ABB RobotStudio station: Laboratorio 1 RS.rspag

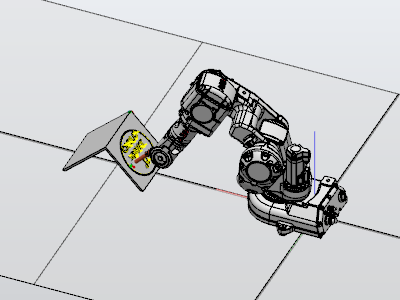
--- station ---
Station Laboratorio 1 RS (saved by RobotStudio 23.2.10395.0)
Controller IRB140_6_81, task T_ROB1: task frame (RAPID world) sits at (164.79, 0, 0) mm in the station
Controller IRB140_6_81
  mechanical unit ROB_1: IRB140_6_81_C_03, 6 joints, base frame (0, 0, 0) mm
Layout (positions relative to the parent item):
  - IRB140_6_81_C_03 [mechanism, from %ABB.RobotStudio.Models.IRB140%\IRB140_6_81_C_G_03.rslib] at (164.79, 0, 0) mm; joint values [0.1988, 0.9588, 0.0809, 3.4211, 0.7525, 2.9948] (rad or m)
  - Tableros [part] at (1000, 0, 0) mm, rotated rx 90 ry 0 rz 180 deg, size 410.4 x 204.7 x 300 mm
  - Marcador [mechanism] at (773, 110, 211.85) mm, rotated rx -180 ry 72.73 rz -180 deg
      TCP MarcadorTCP at (65.54, 0, 135.85) mm, rotated rx 0 ry 25.76 rz 0 deg
      links: EnsambleToolMarcador_3
Attachment: Marcador is attached to IRB140_6_81_C_03 / Link6
Targets, tools, work objects and paths stored in the station and not in the controller backup, written as RAPID:
! task T_ROB1
MODULE Module1
  CONST robtarget Target_350:=[[69.849,197.313,-20],[1,0,0,0],[0,0,0,0],[9E+09,9E+09,9E+09,9E+09,9E+09,9E+09]];
  CONST robtarget Target_360:=[[69.849,197.313,0],[1,0,0,0],[0,0,0,0],[9E+09,9E+09,9E+09,9E+09,9E+09,9E+09]];
  CONST robtarget Target_370:=[[68.877,199.4,0],[1,0,0,0],[0,0,0,0],[9E+09,9E+09,9E+09,9E+09,9E+09,9E+09]];
  CONST robtarget Target_380:=[[67.982,201.773,0],[1,0,0,0],[0,0,0,0],[9E+09,9E+09,9E+09,9E+09,9E+09,9E+09]];
  CONST robtarget Target_390:=[[67.399,204.703,0],[1,0,0,0],[0,0,0,0],[9E+09,9E+09,9E+09,9E+09,9E+09,9E+09]];
  CONST robtarget Target_400:=[[67.178,208.126,0],[1,0,0,0],[0,0,0,0],[9E+09,9E+09,9E+09,9E+09,9E+09,9E+09]];
  CONST robtarget Target_410:=[[71.703,219.575,0],[1,0,0,0],[0,0,0,0],[9E+09,9E+09,9E+09,9E+09,9E+09,9E+09]];
  CONST robtarget Target_420:=[[83.827,223.815,0],[1,0,0,0],[0,0,0,0],[9E+09,9E+09,9E+09,9E+09,9E+09,9E+09]];
  CONST robtarget Target_430:=[[96.066,219.588,0],[1,0,0,0],[0,0,0,0],[9E+09,9E+09,9E+09,9E+09,9E+09,9E+09]];
  CONST robtarget Target_440:=[[100.423,208.152,0],[1,0,0,0],[0,0,0,0],[9E+09,9E+09,9E+09,9E+09,9E+09,9E+09]];
  CONST robtarget Target_450:=[[100.19,204.561,0],[1,0,0,0],[0,0,0,0],[9E+09,9E+09,9E+09,9E+09,9E+09,9E+09]];
  CONST robtarget Target_460:=[[99.489,201.747,0],[1,0,0,0],[0,0,0,0],[9E+09,9E+09,9E+09,9E+09,9E+09,9E+09]];
  CONST robtarget Target_470:=[[98.608,199.348,0],[1,0,0,0],[0,0,0,0],[9E+09,9E+09,9E+09,9E+09,9E+09,9E+09]];
  CONST robtarget Target_480:=[[97.674,197.313,0],[1,0,0,0],[0,0,0,0],[9E+09,9E+09,9E+09,9E+09,9E+09,9E+09]];
  CONST robtarget Target_490:=[[90.154,197.313,0],[1,0,0,0],[0,0,0,0],[9E+09,9E+09,9E+09,9E+09,9E+09,9E+09]];
  CONST robtarget Target_500:=[[90.154,198.039,0],[1,0,0,0],[0,0,0,0],[9E+09,9E+09,9E+09,9E+09,9E+09,9E+09]];
  CONST robtarget Target_510:=[[91.386,199.452,0],[1,0,0,0],[0,0,0,0],[9E+09,9E+09,9E+09,9E+09,9E+09,9E+09]];
  CONST robtarget Target_520:=[[92.721,201.358,0],[1,0,0,0],[0,0,0,0],[9E+09,9E+09,9E+09,9E+09,9E+09,9E+09]];
  CONST robtarget Target_530:=[[93.901,203.783,0],[1,0,0,0],[0,0,0,0],[9E+09,9E+09,9E+09,9E+09,9E+09,9E+09]];
  CONST robtarget Target_540:=[[94.433,206.804,0],[1,0,0,0],[0,0,0,0],[9E+09,9E+09,9E+09,9E+09,9E+09,9E+09]];
  CONST robtarget Target_550:=[[93.901,209.864,0],[1,0,0,0],[0,0,0,0],[9E+09,9E+09,9E+09,9E+09,9E+09,9E+09]];
  CONST robtarget Target_560:=[[92.151,212.639,0],[1,0,0,0],[0,0,0,0],[9E+09,9E+09,9E+09,9E+09,9E+09,9E+09]];
  CONST robtarget Target_570:=[[88.87,214.726,0],[1,0,0,0],[0,0,0,0],[9E+09,9E+09,9E+09,9E+09,9E+09,9E+09]];
  CONST robtarget Target_580:=[[83.852,215.517,0],[1,0,0,0],[0,0,0,0],[9E+09,9E+09,9E+09,9E+09,9E+09,9E+09]];
  CONST robtarget Target_590:=[[78.938,214.752,0],[1,0,0,0],[0,0,0,0],[9E+09,9E+09,9E+09,9E+09,9E+09,9E+09]];
  CONST robtarget Target_600:=[[75.632,212.794,0],[1,0,0,0],[0,0,0,0],[9E+09,9E+09,9E+09,9E+09,9E+09,9E+09]];
  CONST robtarget Target_610:=[[73.713,210.032,0],[1,0,0,0],[0,0,0,0],[9E+09,9E+09,9E+09,9E+09,9E+09,9E+09]];
  CONST robtarget Target_620:=[[73.169,206.856,0],[1,0,0,0],[0,0,0,0],[9E+09,9E+09,9E+09,9E+09,9E+09,9E+09]];
  CONST robtarget Target_630:=[[73.648,204.042,0],[1,0,0,0],[0,0,0,0],[9E+09,9E+09,9E+09,9E+09,9E+09,9E+09]];
  CONST robtarget Target_640:=[[74.828,201.592,0],[1,0,0,0],[0,0,0,0],[9E+09,9E+09,9E+09,9E+09,9E+09,9E+09]];
  CONST robtarget Target_650:=[[76.228,199.595,0],[1,0,0,0],[0,0,0,0],[9E+09,9E+09,9E+09,9E+09,9E+09,9E+09]];
  CONST robtarget Target_660:=[[77.473,198.117,0],[1,0,0,0],[0,0,0,0],[9E+09,9E+09,9E+09,9E+09,9E+09,9E+09]];
  CONST robtarget Target_670:=[[77.473,197.313,0],[1,0,0,0],[0,0,0,0],[9E+09,9E+09,9E+09,9E+09,9E+09,9E+09]];
  CONST robtarget Target_680:=[[69.849,197.313,0],[1,0,0,0],[0,0,0,0],[9E+09,9E+09,9E+09,9E+09,9E+09,9E+09]];
  CONST robtarget Target_690:=[[69.849,197.313,-40],[1,0,0,0],[0,0,0,0],[9E+09,9E+09,9E+09,9E+09,9E+09,9E+09]];
  CONST robtarget Target_850:=[[99.801,165.624,-20],[1,0,0,0],[0,0,0,0],[9E+09,9E+09,9E+09,9E+09,9E+09,9E+09]];
  CONST robtarget Target_860:=[[99.801,165.624,0],[1,0,0,0],[0,0,0,0],[9E+09,9E+09,9E+09,9E+09,9E+09,9E+09]];
  CONST robtarget Target_870:=[[67.801,176.438,0],[1,0,0,0],[0,0,0,0],[9E+09,9E+09,9E+09,9E+09,9E+09,9E+09]];
  CONST robtarget Target_880:=[[67.801,185.203,0],[1,0,0,0],[0,0,0,0],[9E+09,9E+09,9E+09,9E+09,9E+09,9E+09]];
  CONST robtarget Target_890:=[[99.801,196.016,0],[1,0,0,0],[0,0,0,0],[9E+09,9E+09,9E+09,9E+09,9E+09,9E+09]];
  CONST robtarget Target_900:=[[99.801,187.977,0],[1,0,0,0],[0,0,0,0],[9E+09,9E+09,9E+09,9E+09,9E+09,9E+09]];
  CONST robtarget Target_910:=[[93.266,185.955,0],[1,0,0,0],[0,0,0,0],[9E+09,9E+09,9E+09,9E+09,9E+09,9E+09]];
  CONST robtarget Target_920:=[[93.266,175.893,0],[1,0,0,0],[0,0,0,0],[9E+09,9E+09,9E+09,9E+09,9E+09,9E+09]];
  CONST robtarget Target_930:=[[99.801,173.896,0],[1,0,0,0],[0,0,0,0],[9E+09,9E+09,9E+09,9E+09,9E+09,9E+09]];
  CONST robtarget Target_940:=[[99.801,165.624,0],[1,0,0,0],[0,0,0,0],[9E+09,9E+09,9E+09,9E+09,9E+09,9E+09]];
  CONST robtarget Target_950:=[[87.457,177.656,-20],[1,0,0,0],[0,0,0,0],[9E+09,9E+09,9E+09,9E+09,9E+09,9E+09]];
  CONST robtarget Target_960:=[[87.457,177.656,0],[1,0,0,0],[0,0,0,0],[9E+09,9E+09,9E+09,9E+09,9E+09,9E+09]];
  CONST robtarget Target_970:=[[76.877,180.924,0],[1,0,0,0],[0,0,0,0],[9E+09,9E+09,9E+09,9E+09,9E+09,9E+09]];
  CONST robtarget Target_980:=[[87.457,184.217,0],[1,0,0,0],[0,0,0,0],[9E+09,9E+09,9E+09,9E+09,9E+09,9E+09]];
  CONST robtarget Target_990:=[[87.457,177.656,0],[1,0,0,0],[0,0,0,0],[9E+09,9E+09,9E+09,9E+09,9E+09,9E+09]];
  CONST robtarget Target_1000:=[[87.457,177.656,-20],[1,0,0,0],[0,0,0,0],[9E+09,9E+09,9E+09,9E+09,9E+09,9E+09]];
  CONST robtarget Target_1010:=[[99.801,132.872,-20],[1,0,0,0],[0,0,0,0],[9E+09,9E+09,9E+09,9E+09,9E+09,9E+09]];
  CONST robtarget Target_1020:=[[99.801,132.872,0],[1,0,0,0],[0,0,0,0],[9E+09,9E+09,9E+09,9E+09,9E+09,9E+09]];
  CONST robtarget Target_1030:=[[86.186,143.634,0],[1,0,0,0],[0,0,0,0],[9E+09,9E+09,9E+09,9E+09,9E+09,9E+09]];
  CONST robtarget Target_1040:=[[82.543,139.199,0],[1,0,0,0],[0,0,0,0],[9E+09,9E+09,9E+09,9E+09,9E+09,9E+09]];
  CONST robtarget Target_1050:=[[76.592,137.54,0],[1,0,0,0],[0,0,0,0],[9E+09,9E+09,9E+09,9E+09,9E+09,9E+09]];
  CONST robtarget Target_1060:=[[72.3,138.551,0],[1,0,0,0],[0,0,0,0],[9E+09,9E+09,9E+09,9E+09,9E+09,9E+09]];
  CONST robtarget Target_1070:=[[69.512,141.274,0],[1,0,0,0],[0,0,0,0],[9E+09,9E+09,9E+09,9E+09,9E+09,9E+09]];
  CONST robtarget Target_1080:=[[68.138,144.93,0],[1,0,0,0],[0,0,0,0],[9E+09,9E+09,9E+09,9E+09,9E+09,9E+09]];
  CONST robtarget Target_1090:=[[67.801,149.572,0],[1,0,0,0],[0,0,0,0],[9E+09,9E+09,9E+09,9E+09,9E+09,9E+09]];
  CONST robtarget Target_1100:=[[67.801,162.434,0],[1,0,0,0],[0,0,0,0],[9E+09,9E+09,9E+09,9E+09,9E+09,9E+09]];
  CONST robtarget Target_1110:=[[99.801,162.434,0],[1,0,0,0],[0,0,0,0],[9E+09,9E+09,9E+09,9E+09,9E+09,9E+09]];
  CONST robtarget Target_1120:=[[99.801,154.447,0],[1,0,0,0],[0,0,0,0],[9E+09,9E+09,9E+09,9E+09,9E+09,9E+09]];
  CONST robtarget Target_1130:=[[88.053,154.447,0],[1,0,0,0],[0,0,0,0],[9E+09,9E+09,9E+09,9E+09,9E+09,9E+09]];
  CONST robtarget Target_1140:=[[88.053,151.543,0],[1,0,0,0],[0,0,0,0],[9E+09,9E+09,9E+09,9E+09,9E+09,9E+09]];
  CONST robtarget Target_1150:=[[99.801,142.648,0],[1,0,0,0],[0,0,0,0],[9E+09,9E+09,9E+09,9E+09,9E+09,9E+09]];
  CONST robtarget Target_1160:=[[99.801,132.872,0],[1,0,0,0],[0,0,0,0],[9E+09,9E+09,9E+09,9E+09,9E+09,9E+09]];
  CONST robtarget Target_1170:=[[82.297,154.447,-20],[1,0,0,0],[0,0,0,0],[9E+09,9E+09,9E+09,9E+09,9E+09,9E+09]];
  CONST robtarget Target_1180:=[[82.297,154.447,0],[1,0,0,0],[0,0,0,0],[9E+09,9E+09,9E+09,9E+09,9E+09,9E+09]];
  CONST robtarget Target_1190:=[[82.297,152.139,0],[1,0,0,0],[0,0,0,0],[9E+09,9E+09,9E+09,9E+09,9E+09,9E+09]];
  CONST robtarget Target_1200:=[[82.089,149.3,0],[1,0,0,0],[0,0,0,0],[9E+09,9E+09,9E+09,9E+09,9E+09,9E+09]];
  CONST robtarget Target_1210:=[[81.233,147.316,0],[1,0,0,0],[0,0,0,0],[9E+09,9E+09,9E+09,9E+09,9E+09,9E+09]];
  CONST robtarget Target_1220:=[[79.781,146.162,0],[1,0,0,0],[0,0,0,0],[9E+09,9E+09,9E+09,9E+09,9E+09,9E+09]];
  CONST robtarget Target_1230:=[[77.603,145.786,0],[1,0,0,0],[0,0,0,0],[9E+09,9E+09,9E+09,9E+09,9E+09,9E+09]];
  CONST robtarget Target_1240:=[[75.515,146.253,0],[1,0,0,0],[0,0,0,0],[9E+09,9E+09,9E+09,9E+09,9E+09,9E+09]];
  CONST robtarget Target_1250:=[[74.18,147.783,0],[1,0,0,0],[0,0,0,0],[9E+09,9E+09,9E+09,9E+09,9E+09,9E+09]];
  CONST robtarget Target_1260:=[[73.778,149.455,0],[1,0,0,0],[0,0,0,0],[9E+09,9E+09,9E+09,9E+09,9E+09,9E+09]];
  CONST robtarget Target_1270:=[[73.687,151.75,0],[1,0,0,0],[0,0,0,0],[9E+09,9E+09,9E+09,9E+09,9E+09,9E+09]];
  CONST robtarget Target_1280:=[[73.687,154.447,0],[1,0,0,0],[0,0,0,0],[9E+09,9E+09,9E+09,9E+09,9E+09,9E+09]];
  CONST robtarget Target_1290:=[[82.297,154.447,0],[1,0,0,0],[0,0,0,0],[9E+09,9E+09,9E+09,9E+09,9E+09,9E+09]];
  CONST robtarget Target_1300:=[[82.297,154.447,-20],[1,0,0,0],[0,0,0,0],[9E+09,9E+09,9E+09,9E+09,9E+09,9E+09]];
  CONST robtarget Target_1310:=[[99.801,109.144,-20],[1,0,0,0],[0,0,0,0],[9E+09,9E+09,9E+09,9E+09,9E+09,9E+09]];
  CONST robtarget Target_1320:=[[99.801,109.144,0],[1,0,0,0],[0,0,0,0],[9E+09,9E+09,9E+09,9E+09,9E+09,9E+09]];
  CONST robtarget Target_1330:=[[93.707,109.144,0],[1,0,0,0],[0,0,0,0],[9E+09,9E+09,9E+09,9E+09,9E+09,9E+09]];
  CONST robtarget Target_1340:=[[93.707,122.447,0],[1,0,0,0],[0,0,0,0],[9E+09,9E+09,9E+09,9E+09,9E+09,9E+09]];
  CONST robtarget Target_1350:=[[67.801,122.447,0],[1,0,0,0],[0,0,0,0],[9E+09,9E+09,9E+09,9E+09,9E+09,9E+09]];
  CONST robtarget Target_1360:=[[67.801,130.486,0],[1,0,0,0],[0,0,0,0],[9E+09,9E+09,9E+09,9E+09,9E+09,9E+09]];
  CONST robtarget Target_1370:=[[99.801,130.486,0],[1,0,0,0],[0,0,0,0],[9E+09,9E+09,9E+09,9E+09,9E+09,9E+09]];
  CONST robtarget Target_1380:=[[99.801,109.144,0],[1,0,0,0],[0,0,0,0],[9E+09,9E+09,9E+09,9E+09,9E+09,9E+09]];
  CONST robtarget Target_1390:=[[99.801,109.144,-20],[1,0,0,0],[0,0,0,0],[9E+09,9E+09,9E+09,9E+09,9E+09,9E+09]];
  CONST robtarget Target_1400:=[[83.801,76.185,-20],[1,0,0,0],[0,0,0,0],[9E+09,9E+09,9E+09,9E+09,9E+09,9E+09]];
  CONST robtarget Target_1410:=[[83.801,76.185,0],[1,0,0,0],[0,0,0,0],[9E+09,9E+09,9E+09,9E+09,9E+09,9E+09]];
  CONST robtarget Target_1420:=[[96.028,80.334,0],[1,0,0,0],[0,0,0,0],[9E+09,9E+09,9E+09,9E+09,9E+09,9E+09]];
  CONST robtarget Target_1430:=[[100.475,91.692,0],[1,0,0,0],[0,0,0,0],[9E+09,9E+09,9E+09,9E+09,9E+09,9E+09]];
  CONST robtarget Target_1440:=[[95.976,103.05,0],[1,0,0,0],[0,0,0,0],[9E+09,9E+09,9E+09,9E+09,9E+09,9E+09]];
  CONST robtarget Target_1450:=[[83.801,107.173,0],[1,0,0,0],[0,0,0,0],[9E+09,9E+09,9E+09,9E+09,9E+09,9E+09]];
  CONST robtarget Target_1460:=[[71.613,103.05,0],[1,0,0,0],[0,0,0,0],[9E+09,9E+09,9E+09,9E+09,9E+09,9E+09]];
  CONST robtarget Target_1470:=[[67.126,91.692,0],[1,0,0,0],[0,0,0,0],[9E+09,9E+09,9E+09,9E+09,9E+09,9E+09]];
  CONST robtarget Target_1480:=[[71.587,80.334,0],[1,0,0,0],[0,0,0,0],[9E+09,9E+09,9E+09,9E+09,9E+09,9E+09]];
  CONST robtarget Target_1490:=[[83.801,76.185,0],[1,0,0,0],[0,0,0,0],[9E+09,9E+09,9E+09,9E+09,9E+09,9E+09]];
  CONST robtarget Target_1500:=[[75.58,96.671,-20],[1,0,0,0],[0,0,0,0],[9E+09,9E+09,9E+09,9E+09,9E+09,9E+09]];
  CONST robtarget Target_1510:=[[75.58,96.671,0],[1,0,0,0],[0,0,0,0],[9E+09,9E+09,9E+09,9E+09,9E+09,9E+09]];
  CONST robtarget Target_1520:=[[78.887,98.266,0],[1,0,0,0],[0,0,0,0],[9E+09,9E+09,9E+09,9E+09,9E+09,9E+09]];
  CONST robtarget Target_1530:=[[83.801,98.875,0],[1,0,0,0],[0,0,0,0],[9E+09,9E+09,9E+09,9E+09,9E+09,9E+09]];
  CONST robtarget Target_1540:=[[88.702,98.292,0],[1,0,0,0],[0,0,0,0],[9E+09,9E+09,9E+09,9E+09,9E+09,9E+09]];
  CONST robtarget Target_1550:=[[91.969,96.697,0],[1,0,0,0],[0,0,0,0],[9E+09,9E+09,9E+09,9E+09,9E+09,9E+09]];
  CONST robtarget Target_1560:=[[93.862,94.376,0],[1,0,0,0],[0,0,0,0],[9E+09,9E+09,9E+09,9E+09,9E+09,9E+09]];
  CONST robtarget Target_1570:=[[94.433,91.666,0],[1,0,0,0],[0,0,0,0],[9E+09,9E+09,9E+09,9E+09,9E+09,9E+09]];
  CONST robtarget Target_1580:=[[93.823,88.917,0],[1,0,0,0],[0,0,0,0],[9E+09,9E+09,9E+09,9E+09,9E+09,9E+09]];
  CONST robtarget Target_1590:=[[91.917,86.635,5],[1,0,0,0],[0,0,0,0],[9E+09,9E+09,9E+09,9E+09,9E+09,9E+09]];
  CONST robtarget Target_1600:=[[88.663,85.041,0],[1,0,0,0],[0,0,0,0],[9E+09,9E+09,9E+09,9E+09,9E+09,9E+09]];
  CONST robtarget Target_1610:=[[83.801,84.483,0],[1,0,0,0],[0,0,0,0],[9E+09,9E+09,9E+09,9E+09,9E+09,9E+09]];
  CONST robtarget Target_1620:=[[78.912,85.066,0],[1,0,0,0],[0,0,0,0],[9E+09,9E+09,9E+09,9E+09,9E+09,9E+09]];
  CONST robtarget Target_1630:=[[75.632,86.661,0],[1,0,0,0],[0,0,0,0],[9E+09,9E+09,9E+09,9E+09,9E+09,9E+09]];
  CONST robtarget Target_1640:=[[73.739,88.969,0],[1,0,0,0],[0,0,0,0],[9E+09,9E+09,9E+09,9E+09,9E+09,9E+09]];
  CONST robtarget Target_1650:=[[73.169,91.666,0],[1,0,0,0],[0,0,0,0],[9E+09,9E+09,9E+09,9E+09,9E+09,9E+09]];
  CONST robtarget Target_1660:=[[73.7,94.35,0],[1,0,0,0],[0,0,0,0],[9E+09,9E+09,9E+09,9E+09,9E+09,9E+09]];
  CONST robtarget Target_1670:=[[75.58,96.671,0],[1,0,0,0],[0,0,0,0],[9E+09,9E+09,9E+09,9E+09,9E+09,9E+09]];
  CONST robtarget Target_1680:=[[75.58,96.671,-20],[1,0,0,0],[0,0,0,0],[9E+09,9E+09,9E+09,9E+09,9E+09,9E+09]];
  CONST robtarget Target_1690:=[[120.488,219.705,-20],[1,0,0,0],[0,0,0,0],[9E+09,9E+09,9E+09,9E+09,9E+09,9E+09]];
  CONST robtarget Target_1700:=[[120.488,219.705,0],[1,0,0,0],[0,0,0,0],[9E+09,9E+09,9E+09,9E+09,9E+09,9E+09]];
  CONST robtarget Target_1710:=[[120.488,204.353,0],[1,0,0,0],[0,0,0,0],[9E+09,9E+09,9E+09,9E+09,9E+09,9E+09]];
  CONST robtarget Target_1720:=[[143.1,204.353,0.001],[1,0,0,0],[0,0,0,0],[9E+09,9E+09,9E+09,9E+09,9E+09,9E+09]];
  CONST robtarget Target_1730:=[[147.016,205.066,0.001],[1,0,0,0],[0,0,0,0],[9E+09,9E+09,9E+09,9E+09,9E+09,9E+09]];
  CONST robtarget Target_1740:=[[150.154,207.206,0.001],[1,0,0,0],[0,0,0,0],[9E+09,9E+09,9E+09,9E+09,9E+09,9E+09]];
  CONST robtarget Target_1750:=[[152.293,211.005,0.001],[1,0,0,0],[0,0,0,0],[9E+09,9E+09,9E+09,9E+09,9E+09,9E+09]];
  CONST robtarget Target_1760:=[[152.98,216.049,0.001],[1,0,0,0],[0,0,0,0],[9E+09,9E+09,9E+09,9E+09,9E+09,9E+09]];
  CONST robtarget Target_1770:=[[152.825,220.042,0.001],[1,0,0,0],[0,0,0,0],[9E+09,9E+09,9E+09,9E+09,9E+09,9E+09]];
  CONST robtarget Target_1780:=[[152.358,223.335,0.001],[1,0,0,0],[0,0,0,0],[9E+09,9E+09,9E+09,9E+09,9E+09,9E+09]];
  CONST robtarget Target_1790:=[[145.875,223.335,0.001],[1,0,0,0],[0,0,0,0],[9E+09,9E+09,9E+09,9E+09,9E+09,9E+09]];
  CONST robtarget Target_1800:=[[146.601,220.6,0.001],[1,0,0,0],[0,0,0,0],[9E+09,9E+09,9E+09,9E+09,9E+09,9E+09]];
  CONST robtarget Target_1810:=[[146.938,217.89,0.001],[1,0,0,0],[0,0,0,0],[9E+09,9E+09,9E+09,9E+09,9E+09,9E+09]];
  CONST robtarget Target_1820:=[[146.342,214.609,0.001],[1,0,0,0],[0,0,0,0],[9E+09,9E+09,9E+09,9E+09,9E+09,9E+09]];
  CONST robtarget Target_1830:=[[144.656,212.989,0.001],[1,0,0,0],[0,0,0,0],[9E+09,9E+09,9E+09,9E+09,9E+09,9E+09]];
  CONST robtarget Target_1840:=[[142.219,212.444,0.001],[1,0,0,0],[0,0,0,0],[9E+09,9E+09,9E+09,9E+09,9E+09,9E+09]];
  CONST robtarget Target_1850:=[[139.133,212.392,0],[1,0,0,0],[0,0,0,0],[9E+09,9E+09,9E+09,9E+09,9E+09,9E+09]];
  CONST robtarget Target_1860:=[[126.297,212.392,0],[1,0,0,0],[0,0,0,0],[9E+09,9E+09,9E+09,9E+09,9E+09,9E+09]];
  CONST robtarget Target_1870:=[[126.297,219.705,0],[1,0,0,0],[0,0,0,0],[9E+09,9E+09,9E+09,9E+09,9E+09,9E+09]];
  CONST robtarget Target_1880:=[[120.488,219.705,0],[1,0,0,0],[0,0,0,0],[9E+09,9E+09,9E+09,9E+09,9E+09,9E+09]];
  CONST robtarget Target_1890:=[[120.488,219.705,-20],[1,0,0,0],[0,0,0,0],[9E+09,9E+09,9E+09,9E+09,9E+09,9E+09]];
  CONST robtarget Target_1900:=[[153.162,184.515,-20],[1,0,0,0],[0,0,0,0],[9E+09,9E+09,9E+09,9E+09,9E+09,9E+09]];
  CONST robtarget Target_1910:=[[153.162,184.515,0],[1,0,0,0],[0,0,0,0],[9E+09,9E+09,9E+09,9E+09,9E+09,9E+09]];
  CONST robtarget Target_1920:=[[148.715,173.157,0.001],[1,0,0,0],[0,0,0,0],[9E+09,9E+09,9E+09,9E+09,9E+09,9E+09]];
  CONST robtarget Target_1930:=[[136.488,169.008,0],[1,0,0,0],[0,0,0,0],[9E+09,9E+09,9E+09,9E+09,9E+09,9E+09]];
  CONST robtarget Target_1940:=[[124.274,173.157,0],[1,0,0,0],[0,0,0,0],[9E+09,9E+09,9E+09,9E+09,9E+09,9E+09]];
  CONST robtarget Target_1950:=[[119.814,184.515,0],[1,0,0,0],[0,0,0,0],[9E+09,9E+09,9E+09,9E+09,9E+09,9E+09]];
  CONST robtarget Target_1960:=[[124.3,195.874,0],[1,0,0,0],[0,0,0,0],[9E+09,9E+09,9E+09,9E+09,9E+09,9E+09]];
  CONST robtarget Target_1970:=[[136.488,199.997,0],[1,0,0,0],[0,0,0,0],[9E+09,9E+09,9E+09,9E+09,9E+09,9E+09]];
  CONST robtarget Target_1980:=[[148.663,195.874,0.001],[1,0,0,0],[0,0,0,0],[9E+09,9E+09,9E+09,9E+09,9E+09,9E+09]];
  CONST robtarget Target_1990:=[[153.162,184.515,0.001],[1,0,0,0],[0,0,0,0],[9E+09,9E+09,9E+09,9E+09,9E+09,9E+09]];
  CONST robtarget Target_2000:=[[144.604,179.459,-20],[1,0,0,0],[0,0,0,0],[9E+09,9E+09,9E+09,9E+09,9E+09,9E+09]];
  CONST robtarget Target_2010:=[[144.604,179.459,0.001],[1,0,0,0],[0,0,0,0],[9E+09,9E+09,9E+09,9E+09,9E+09,9E+09]];
  CONST robtarget Target_2020:=[[141.35,177.864,0.001],[1,0,0,0],[0,0,0,0],[9E+09,9E+09,9E+09,9E+09,9E+09,9E+09]];
  CONST robtarget Target_2030:=[[136.488,177.306,0],[1,0,0,0],[0,0,0,0],[9E+09,9E+09,9E+09,9E+09,9E+09,9E+09]];
  CONST robtarget Target_2040:=[[131.6,177.89,0],[1,0,0,0],[0,0,0,0],[9E+09,9E+09,9E+09,9E+09,9E+09,9E+09]];
  CONST robtarget Target_2050:=[[128.319,179.485,0],[1,0,0,0],[0,0,0,0],[9E+09,9E+09,9E+09,9E+09,9E+09,9E+09]];
  CONST robtarget Target_2060:=[[126.426,181.793,0],[1,0,0,0],[0,0,0,0],[9E+09,9E+09,9E+09,9E+09,9E+09,9E+09]];
  CONST robtarget Target_2070:=[[125.856,184.489,0],[1,0,0,0],[0,0,0,0],[9E+09,9E+09,9E+09,9E+09,9E+09,9E+09]];
  CONST robtarget Target_2080:=[[126.387,187.173,0],[1,0,0,0],[0,0,0,0],[9E+09,9E+09,9E+09,9E+09,9E+09,9E+09]];
  CONST robtarget Target_2090:=[[128.267,189.494,0],[1,0,0,0],[0,0,0,0],[9E+09,9E+09,9E+09,9E+09,9E+09,9E+09]];
  CONST robtarget Target_2100:=[[131.574,191.089,0],[1,0,0,0],[0,0,0,0],[9E+09,9E+09,9E+09,9E+09,9E+09,9E+09]];
  CONST robtarget Target_2110:=[[136.488,191.699,0],[1,0,0,0],[0,0,0,0],[9E+09,9E+09,9E+09,9E+09,9E+09,9E+09]];
  CONST robtarget Target_2120:=[[141.389,191.115,0.001],[1,0,0,0],[0,0,0,0],[9E+09,9E+09,9E+09,9E+09,9E+09,9E+09]];
  CONST robtarget Target_2130:=[[144.656,189.52,0.001],[1,0,0,0],[0,0,0,0],[9E+09,9E+09,9E+09,9E+09,9E+09,9E+09]];
  CONST robtarget Target_2140:=[[146.549,187.199,0.001],[1,0,0,0],[0,0,0,0],[9E+09,9E+09,9E+09,9E+09,9E+09,9E+09]];
  CONST robtarget Target_2150:=[[147.12,184.489,0.001],[1,0,0,0],[0,0,0,0],[9E+09,9E+09,9E+09,9E+09,9E+09,9E+09]];
  CONST robtarget Target_2160:=[[146.51,181.741,0.001],[1,0,0,0],[0,0,0,0],[9E+09,9E+09,9E+09,9E+09,9E+09,9E+09]];
  CONST robtarget Target_2170:=[[144.604,179.459,0.001],[1,0,0,0],[0,0,0,0],[9E+09,9E+09,9E+09,9E+09,9E+09,9E+09]];
  CONST robtarget Target_2180:=[[144.604,179.459,-20],[1,0,0,0],[0,0,0,0],[9E+09,9E+09,9E+09,9E+09,9E+09,9E+09]];
  CONST robtarget Target_2190:=[[152.488,136.827,-20],[1,0,0,0],[0,0,0,0],[9E+09,9E+09,9E+09,9E+09,9E+09,9E+09]];
  CONST robtarget Target_2200:=[[152.488,136.827,0.001],[1,0,0,0],[0,0,0,0],[9E+09,9E+09,9E+09,9E+09,9E+09,9E+09]];
  CONST robtarget Target_2210:=[[120.488,136.827,0],[1,0,0,0],[0,0,0,0],[9E+09,9E+09,9E+09,9E+09,9E+09,9E+09]];
  CONST robtarget Target_2220:=[[120.488,144.165,0],[1,0,0,0],[0,0,0,0],[9E+09,9E+09,9E+09,9E+09,9E+09,9E+09]];
  CONST robtarget Target_2230:=[[138.822,144.165,0],[1,0,0,0],[0,0,0,0],[9E+09,9E+09,9E+09,9E+09,9E+09,9E+09]];
  CONST robtarget Target_2240:=[[120.488,154.382,0],[1,0,0,0],[0,0,0,0],[9E+09,9E+09,9E+09,9E+09,9E+09,9E+09]];
  CONST robtarget Target_2250:=[[120.488,164.237,0],[1,0,0,0],[0,0,0,0],[9E+09,9E+09,9E+09,9E+09,9E+09,9E+09]];
  CONST robtarget Target_2260:=[[152.488,164.237,0.001],[1,0,0,0],[0,0,0,0],[9E+09,9E+09,9E+09,9E+09,9E+09,9E+09]];
  CONST robtarget Target_2270:=[[152.488,156.898,0.001],[1,0,0,0],[0,0,0,0],[9E+09,9E+09,9E+09,9E+09,9E+09,9E+09]];
  CONST robtarget Target_2280:=[[130.186,156.898,0],[1,0,0,0],[0,0,0,0],[9E+09,9E+09,9E+09,9E+09,9E+09,9E+09]];
  CONST robtarget Target_2290:=[[152.488,144.554,0.001],[1,0,0,0],[0,0,0,0],[9E+09,9E+09,9E+09,9E+09,9E+09,9E+09]];
  CONST robtarget Target_2300:=[[152.488,136.827,0.001],[1,0,0,0],[0,0,0,0],[9E+09,9E+09,9E+09,9E+09,9E+09,9E+09]];
  CONST robtarget Target_2310:=[[152.488,136.827,-20],[1,0,0,0],[0,0,0,0],[9E+09,9E+09,9E+09,9E+09,9E+09,9E+09]];
  CONST robtarget Target_2320:=[[152.488,103.374,-20],[1,0,0,0],[0,0,0,0],[9E+09,9E+09,9E+09,9E+09,9E+09,9E+09]];
  CONST robtarget Target_2330:=[[152.488,103.374,0.001],[1,0,0,0],[0,0,0,0],[9E+09,9E+09,9E+09,9E+09,9E+09,9E+09]];
  CONST robtarget Target_2340:=[[120.488,114.188,0],[1,0,0,0],[0,0,0,0],[9E+09,9E+09,9E+09,9E+09,9E+09,9E+09]];
  CONST robtarget Target_2350:=[[120.488,122.953,0],[1,0,0,0],[0,0,0,0],[9E+09,9E+09,9E+09,9E+09,9E+09,9E+09]];
  CONST robtarget Target_2360:=[[152.488,133.767,0.001],[1,0,0,0],[0,0,0,0],[9E+09,9E+09,9E+09,9E+09,9E+09,9E+09]];
  CONST robtarget Target_2370:=[[152.488,125.728,0.001],[1,0,0,0],[0,0,0,0],[9E+09,9E+09,9E+09,9E+09,9E+09,9E+09]];
  CONST robtarget Target_2380:=[[145.953,123.705,0.001],[1,0,0,0],[0,0,0,0],[9E+09,9E+09,9E+09,9E+09,9E+09,9E+09]];
  CONST robtarget Target_2390:=[[145.953,113.643,0.001],[1,0,0,0],[0,0,0,0],[9E+09,9E+09,9E+09,9E+09,9E+09,9E+09]];
  CONST robtarget Target_2400:=[[152.488,111.647,0.001],[1,0,0,0],[0,0,0,0],[9E+09,9E+09,9E+09,9E+09,9E+09,9E+09]];
  CONST robtarget Target_2410:=[[152.488,103.374,0.001],[1,0,0,0],[0,0,0,0],[9E+09,9E+09,9E+09,9E+09,9E+09,9E+09]];
  CONST robtarget Target_2420:=[[140.144,115.407,-20],[1,0,0,0],[0,0,0,0],[9E+09,9E+09,9E+09,9E+09,9E+09,9E+09]];
  CONST robtarget Target_2430:=[[140.144,115.407,0.001],[1,0,0,0],[0,0,0,0],[9E+09,9E+09,9E+09,9E+09,9E+09,9E+09]];
  CONST robtarget Target_2440:=[[129.564,118.674,0],[1,0,0,0],[0,0,0,0],[9E+09,9E+09,9E+09,9E+09,9E+09,9E+09]];
  CONST robtarget Target_2450:=[[140.144,121.968,0.001],[1,0,0,0],[0,0,0,0],[9E+09,9E+09,9E+09,9E+09,9E+09,9E+09]];
  CONST robtarget Target_2460:=[[140.144,115.407,0.001],[1,0,0,0],[0,0,0,0],[9E+09,9E+09,9E+09,9E+09,9E+09,9E+09]];
  CONST robtarget Target_2470:=[[140.144,115.407,-20],[1,0,0,0],[0,0,0,0],[9E+09,9E+09,9E+09,9E+09,9E+09,9E+09]];
  CONST robtarget Target_2480:=[[152.488,86,-20],[1,0,0,0],[0,0,0,0],[9E+09,9E+09,9E+09,9E+09,9E+09,9E+09]];
  CONST robtarget Target_2490:=[[152.488,86,0.001],[1,0,0,0],[0,0,0,0],[9E+09,9E+09,9E+09,9E+09,9E+09,9E+09]];
  CONST robtarget Target_2500:=[[126.582,86,0],[1,0,0,0],[0,0,0,0],[9E+09,9E+09,9E+09,9E+09,9E+09,9E+09]];
  CONST robtarget Target_2510:=[[126.582,76.535,0],[1,0,0,0],[0,0,0,0],[9E+09,9E+09,9E+09,9E+09,9E+09,9E+09]];
  CONST robtarget Target_2520:=[[120.488,76.535,0],[1,0,0,0],[0,0,0,0],[9E+09,9E+09,9E+09,9E+09,9E+09,9E+09]];
  CONST robtarget Target_2530:=[[120.488,103.504,0],[1,0,0,0],[0,0,0,0],[9E+09,9E+09,9E+09,9E+09,9E+09,9E+09]];
  CONST robtarget Target_2540:=[[126.582,103.504,0],[1,0,0,0],[0,0,0,0],[9E+09,9E+09,9E+09,9E+09,9E+09,9E+09]];
  CONST robtarget Target_2550:=[[126.582,94.039,0],[1,0,0,0],[0,0,0,0],[9E+09,9E+09,9E+09,9E+09,9E+09,9E+09]];
  CONST robtarget Target_2560:=[[152.488,94.039,0.001],[1,0,0,0],[0,0,0,0],[9E+09,9E+09,9E+09,9E+09,9E+09,9E+09]];
  CONST robtarget Target_2570:=[[152.488,86,0.001],[1,0,0,0],[0,0,0,0],[9E+09,9E+09,9E+09,9E+09,9E+09,9E+09]];
  CONST robtarget Target_2580:=[[152.488,86,-20],[1,0,0,0],[0,0,0,0],[9E+09,9E+09,9E+09,9E+09,9E+09,9E+09]];
  CONST robtarget Target_2590:=[[210.888,134.542,-20],[1,0,0,0],[0,0,0,0],[9E+09,9E+09,9E+09,9E+09,9E+09,9E+09]];
  CONST robtarget Target_2600:=[[210.888,134.542,0.001],[1,0,0,0],[0,0,0,0],[9E+09,9E+09,9E+09,9E+09,9E+09,9E+09]];
  CONST robtarget Target_2610:=[[186.577,134.542,0.001],[1,0,0,0],[0,0,0,0],[9E+09,9E+09,9E+09,9E+09,9E+09,9E+09]];
  CONST robtarget Target_2620:=[[192.776,154.518,0.001],[1,0,0,0],[0,0,0,0],[9E+09,9E+09,9E+09,9E+09,9E+09,9E+09]];
  CONST robtarget Target_2630:=[[220.856,154.518,0.001],[1,0,0,0],[0,0,0,0],[9E+09,9E+09,9E+09,9E+09,9E+09,9E+09]];
  CONST robtarget Target_2640:=[[229.253,157.086,0.001],[1,0,0,0],[0,0,0,0],[9E+09,9E+09,9E+09,9E+09,9E+09,9E+09]];
  CONST robtarget Target_2650:=[[232.16,165.012,0.001],[1,0,0,0],[0,0,0,0],[9E+09,9E+09,9E+09,9E+09,9E+09,9E+09]];
  CONST robtarget Target_2660:=[[230.094,170.806,0.001],[1,0,0,0],[0,0,0,0],[9E+09,9E+09,9E+09,9E+09,9E+09,9E+09]];
  CONST robtarget Target_2670:=[[224.705,172.954,0.001],[1,0,0,0],[0,0,0,0],[9E+09,9E+09,9E+09,9E+09,9E+09,9E+09]];
  CONST robtarget Target_2680:=[[218.789,170.401,0.001],[1,0,0,0],[0,0,0,0],[9E+09,9E+09,9E+09,9E+09,9E+09,9E+09]];
  CONST robtarget Target_2690:=[[216.399,163.716,0.001],[1,0,0,0],[0,0,0,0],[9E+09,9E+09,9E+09,9E+09,9E+09,9E+09]];
  CONST robtarget Target_2700:=[[216.784,160.94,0.001],[1,0,0,0],[0,0,0,0],[9E+09,9E+09,9E+09,9E+09,9E+09,9E+09]];
  CONST robtarget Target_2710:=[[217.938,157.881,0.001],[1,0,0,0],[0,0,0,0],[9E+09,9E+09,9E+09,9E+09,9E+09,9E+09]];
  CONST robtarget Target_2720:=[[185.159,157.881,0.001],[1,0,0,0],[0,0,0,0],[9E+09,9E+09,9E+09,9E+09,9E+09,9E+09]];
  CONST robtarget Target_2730:=[[176.852,131.139,0.001],[1,0,0,0],[0,0,0,0],[9E+09,9E+09,9E+09,9E+09,9E+09,9E+09]];
  CONST robtarget Target_2740:=[[214.048,131.139,0.001],[1,0,0,0],[0,0,0,0],[9E+09,9E+09,9E+09,9E+09,9E+09,9E+09]];
  CONST robtarget Target_2750:=[[222.254,133.615,0.001],[1,0,0,0],[0,0,0,0],[9E+09,9E+09,9E+09,9E+09,9E+09,9E+09]];
  CONST robtarget Target_2760:=[[225.191,141.511,0.001],[1,0,0,0],[0,0,0,0],[9E+09,9E+09,9E+09,9E+09,9E+09,9E+09]];
  CONST robtarget Target_2770:=[[223.084,147.346,0.001],[1,0,0,0],[0,0,0,0],[9E+09,9E+09,9E+09,9E+09,9E+09,9E+09]];
  CONST robtarget Target_2780:=[[217.655,149.534,0.001],[1,0,0,0],[0,0,0,0],[9E+09,9E+09,9E+09,9E+09,9E+09,9E+09]];
  CONST robtarget Target_2790:=[[211.86,146.941,0.001],[1,0,0,0],[0,0,0,0],[9E+09,9E+09,9E+09,9E+09,9E+09,9E+09]];
  CONST robtarget Target_2800:=[[209.429,140.255,0.001],[1,0,0,0],[0,0,0,0],[9E+09,9E+09,9E+09,9E+09,9E+09,9E+09]];
  CONST robtarget Target_2810:=[[209.672,137.905,0.001],[1,0,0,0],[0,0,0,0],[9E+09,9E+09,9E+09,9E+09,9E+09,9E+09]];
  CONST robtarget Target_2820:=[[210.888,134.542,0.001],[1,0,0,0],[0,0,0,0],[9E+09,9E+09,9E+09,9E+09,9E+09,9E+09]];
  CONST robtarget Target_2830:=[[210.888,134.542,-20],[1,0,0,0],[0,0,0,0],[9E+09,9E+09,9E+09,9E+09,9E+09,9E+09]];
  CONST robtarget Target_2890:=[[149.643,260,-20],[1,0,0,0],[0,0,0,0],[9E+09,9E+09,9E+09,9E+09,9E+09,9E+09]];
  CONST robtarget Target_2900:=[[149.643,260,0.001],[1,0,0,0],[0,0,0,0],[9E+09,9E+09,9E+09,9E+09,9E+09,9E+09]];
  CONST robtarget Target_2910:=[[43.169,122.373,0],[1,0,0,0],[0,0,0,0],[9E+09,9E+09,9E+09,9E+09,9E+09,9E+09]];
  CONST robtarget Target_2920:=[[149.643,40,0.001],[1,0,0,0],[0,0,0,0],[9E+09,9E+09,9E+09,9E+09,9E+09,9E+09]];
  CONST robtarget Target_2930:=[[258.691,135.554,0.001],[1,0,0,0],[0,0,0,0],[9E+09,9E+09,9E+09,9E+09,9E+09,9E+09]];
  CONST robtarget Target_2940:=[[149.643,260,0.001],[1,0,0,0],[0,0,0,0],[9E+09,9E+09,9E+09,9E+09,9E+09,9E+09]];
  CONST robtarget Target_2950:=[[149.643,260,-20],[1,0,0,0],[0,0,0,0],[9E+09,9E+09,9E+09,9E+09,9E+09,9E+09]];
  PROC Path_1C()
    MoveJ Target_350,v200,z10,tool0\WObj:=Tableros;
    MoveL Target_360,v100,z0,tool0\WObj:=Tableros;
    MoveC Target_370,Target_380,v100,z0,tool0\WObj:=Tableros;
    MoveC Target_390,Target_400,v100,z0,tool0\WObj:=Tableros;
    MoveC Target_410,Target_420,v100,z0,tool0\WObj:=Tableros;
    MoveC Target_430,Target_440,v100,z0,tool0\WObj:=Tableros;
    MoveC Target_450,Target_460,v100,z0,tool0\WObj:=Tableros;
    MoveC Target_470,Target_480,v100,z0,tool0\WObj:=Tableros;
    MoveL Target_490,v100,z0,tool0\WObj:=Tableros;
    MoveL Target_500,v100,z0,tool0\WObj:=Tableros;
    MoveC Target_510,Target_520,v100,z0,tool0\WObj:=Tableros;
    MoveC Target_530,Target_540,v100,z0,tool0\WObj:=Tableros;
    MoveC Target_550,Target_560,v100,z0,tool0\WObj:=Tableros;
    MoveC Target_570,Target_580,v100,z0,tool0\WObj:=Tableros;
    MoveC Target_590,Target_600,v100,z0,tool0\WObj:=Tableros;
    MoveC Target_610,Target_620,v100,z0,tool0\WObj:=Tableros;
    MoveC Target_630,Target_640,v100,z0,tool0\WObj:=Tableros;
    MoveC Target_650,Target_660,v100,z0,tool0\WObj:=Tableros;
    MoveL Target_670,v100,z0,tool0\WObj:=Tableros;
    MoveL Target_680,v100,z0,tool0\WObj:=Tableros;
    MoveL Target_690,v100,z0,tool0\WObj:=Tableros;
  ENDPROC
  PROC Path_1A()
    MoveJ Target_850,v100,z10,tool0\WObj:=Tableros;
    MoveL Target_860,v100,z0,tool0\WObj:=Tableros;
    MoveL Target_870,v100,z0,tool0\WObj:=Tableros;
    MoveL Target_880,v100,z0,tool0\WObj:=Tableros;
    MoveL Target_890,v100,z0,tool0\WObj:=Tableros;
    MoveL Target_900,v100,z0,tool0\WObj:=Tableros;
    MoveL Target_910,v100,z0,tool0\WObj:=Tableros;
    MoveL Target_920,v100,z0,tool0\WObj:=Tableros;
    MoveL Target_930,v100,z0,tool0\WObj:=Tableros;
    MoveL Target_940,v100,z0,tool0\WObj:=Tableros;
    MoveL Target_950,v100,z0,tool0\WObj:=Tableros;
    MoveL Target_960,v100,z0,tool0\WObj:=Tableros;
    MoveL Target_970,v100,z0,tool0\WObj:=Tableros;
    MoveL Target_980,v100,z0,tool0\WObj:=Tableros;
    MoveL Target_990,v100,z0,tool0\WObj:=Tableros;
    MoveL Target_1000,v100,z0,tool0\WObj:=Tableros;
  ENDPROC
  PROC Path_1R()
    MoveJ Target_1010,v200,z10,tool0\WObj:=Tableros;
    MoveL Target_1020,v100,z0,tool0\WObj:=Tableros;
    MoveL Target_1030,v100,z0,tool0\WObj:=Tableros;
    MoveC Target_1040,Target_1050,v100,z0,tool0\WObj:=Tableros;
    MoveC Target_1060,Target_1070,v100,z0,tool0\WObj:=Tableros;
    MoveC Target_1080,Target_1090,v100,z0,tool0\WObj:=Tableros;
    MoveL Target_1100,v100,z0,tool0\WObj:=Tableros;
    MoveL Target_1110,v100,z0,tool0\WObj:=Tableros;
    MoveL Target_1120,v100,z0,tool0\WObj:=Tableros;
    MoveL Target_1130,v100,z0,tool0\WObj:=Tableros;
    MoveL Target_1140,v100,z0,tool0\WObj:=Tableros;
    MoveL Target_1150,v100,z0,tool0\WObj:=Tableros;
    MoveL Target_1160,v100,z0,tool0\WObj:=Tableros;
    MoveL Target_1170,v100,z0,tool0\WObj:=Tableros;
    MoveL Target_1180,v100,z0,tool0\WObj:=Tableros;
    MoveL Target_1190,v100,z0,tool0\WObj:=Tableros;
    MoveC Target_1200,Target_1210,v100,z0,tool0\WObj:=Tableros;
    MoveC Target_1220,Target_1230,v100,z0,tool0\WObj:=Tableros;
    MoveC Target_1240,Target_1250,v100,z0,tool0\WObj:=Tableros;
    MoveC Target_1260,Target_1270,v100,z0,tool0\WObj:=Tableros;
    MoveL Target_1280,v100,z0,tool0\WObj:=Tableros;
    MoveL Target_1290,v100,z0,tool0\WObj:=Tableros;
    MoveL Target_1300,v100,z0,tool0\WObj:=Tableros;
  ENDPROC
  PROC Path_1L()
    MoveJ Target_1310,v200,z10,tool0\WObj:=Tableros;
    MoveL Target_1320,v100,z0,tool0\WObj:=Tableros;
    MoveL Target_1330,v100,z0,tool0\WObj:=Tableros;
    MoveL Target_1340,v100,z0,tool0\WObj:=Tableros;
    MoveL Target_1350,v100,z0,tool0\WObj:=Tableros;
    MoveL Target_1360,v100,z0,tool0\WObj:=Tableros;
    MoveL Target_1370,v100,z0,tool0\WObj:=Tableros;
    MoveL Target_1380,v100,z0,tool0\WObj:=Tableros;
    MoveL Target_1390,v100,z0,tool0\WObj:=Tableros;
  ENDPROC
  PROC Path_1O()
    MoveJ Target_1400,v200,z10,MarcadorTCP\WObj:=Tableros;
    MoveL Target_1410,v100,z10,MarcadorTCP\WObj:=Tableros;
    MoveC Target_1420,Target_1430,v100,z10,MarcadorTCP\WObj:=Tableros;
    MoveC Target_1440,Target_1450,v100,z10,MarcadorTCP\WObj:=Tableros;
    MoveC Target_1460,Target_1470,v100,z10,MarcadorTCP\WObj:=Tableros;
    MoveC Target_1480,Target_1490,v100,z10,MarcadorTCP\WObj:=Tableros;
    MoveL Target_1500,v100,z10,MarcadorTCP\WObj:=Tableros;
    MoveL Target_1510,v100,z10,MarcadorTCP\WObj:=Tableros;
    MoveC Target_1520,Target_1530,v100,z10,MarcadorTCP\WObj:=Tableros;
    MoveC Target_1540,Target_1550,v100,z10,MarcadorTCP\WObj:=Tableros;
    MoveC Target_1560,Target_1570,v100,z10,MarcadorTCP\WObj:=Tableros;
    MoveC Target_1580,Target_1590,v100,z10,MarcadorTCP\WObj:=Tableros;
    MoveC Target_1600,Target_1610,v100,z10,MarcadorTCP\WObj:=Tableros;
    MoveC Target_1620,Target_1630,v100,z10,MarcadorTCP\WObj:=Tableros;
    MoveC Target_1640,Target_1650,v100,z10,MarcadorTCP\WObj:=Tableros;
    MoveC Target_1660,Target_1670,v100,z10,MarcadorTCP\WObj:=Tableros;
    MoveL Target_1680,v100,z10,MarcadorTCP\WObj:=Tableros;
  ENDPROC
  PROC Path_2J()
    MoveL Target_1690,v100,z0,tool0\WObj:=Tableros;
    MoveL Target_1700,v100,z0,tool0\WObj:=Tableros;
    MoveL Target_1710,v100,z0,tool0\WObj:=Tableros;
    MoveL Target_1720,v100,z0,tool0\WObj:=Tableros;
    MoveC Target_1730,Target_1740,v100,z0,tool0\WObj:=Tableros;
    MoveC Target_1750,Target_1760,v100,z0,tool0\WObj:=Tableros;
    MoveC Target_1770,Target_1780,v100,z0,tool0\WObj:=Tableros;
    MoveL Target_1790,v100,z0,tool0\WObj:=Tableros;
    MoveC Target_1800,Target_1810,v100,z0,tool0\WObj:=Tableros;
    MoveC Target_1820,Target_1830,v100,z0,tool0\WObj:=Tableros;
    MoveC Target_1840,Target_1850,v100,z0,tool0\WObj:=Tableros;
    MoveL Target_1860,v100,z0,tool0\WObj:=Tableros;
    MoveL Target_1870,v100,z0,tool0\WObj:=Tableros;
    MoveL Target_1880,v100,z0,tool0\WObj:=Tableros;
    MoveL Target_1890,v100,z0,tool0\WObj:=Tableros;
  ENDPROC
  PROC Path_2O()
    MoveL Target_1900,v100,z0,tool0\WObj:=Tableros;
    MoveL Target_1910,v100,z0,tool0\WObj:=Tableros;
    MoveC Target_1920,Target_1930,v100,z0,tool0\WObj:=Tableros;
    MoveC Target_1940,Target_1950,v100,z0,tool0\WObj:=Tableros;
    MoveC Target_1960,Target_1970,v100,z0,tool0\WObj:=Tableros;
    MoveC Target_1980,Target_1990,v100,z0,tool0\WObj:=Tableros;
    MoveL Target_2000,v100,z0,tool0\WObj:=Tableros;
    MoveL Target_2010,v100,z0,tool0\WObj:=Tableros;
    MoveC Target_2020,Target_2030,v100,z0,tool0\WObj:=Tableros;
    MoveC Target_2040,Target_2050,v100,z0,tool0\WObj:=Tableros;
    MoveC Target_2060,Target_2070,v100,z0,tool0\WObj:=Tableros;
    MoveC Target_2080,Target_2090,v100,z0,tool0\WObj:=Tableros;
    MoveC Target_2100,Target_2110,v100,z0,tool0\WObj:=Tableros;
    MoveC Target_2120,Target_2130,v100,z0,tool0\WObj:=Tableros;
    MoveC Target_2140,Target_2150,v100,z0,tool0\WObj:=Tableros;
    MoveC Target_2160,Target_2170,v100,z0,tool0\WObj:=Tableros;
    MoveL Target_2180,v100,z0,tool0\WObj:=Tableros;
  ENDPROC
  PROC Path_2N()
    MoveJ Target_2190,v200,z10,tool0\WObj:=Tableros;
    MoveL Target_2200,v100,z0,tool0\WObj:=Tableros;
    MoveL Target_2210,v100,z0,tool0\WObj:=Tableros;
    MoveL Target_2220,v100,z0,tool0\WObj:=Tableros;
    MoveL Target_2230,v100,z0,tool0\WObj:=Tableros;
    MoveL Target_2240,v100,z0,tool0\WObj:=Tableros;
    MoveL Target_2250,v100,z0,tool0\WObj:=Tableros;
    MoveL Target_2260,v100,z0,tool0\WObj:=Tableros;
    MoveL Target_2270,v100,z0,tool0\WObj:=Tableros;
    MoveL Target_2280,v100,z0,tool0\WObj:=Tableros;
    MoveL Target_2290,v100,z0,tool0\WObj:=Tableros;
    MoveL Target_2300,v100,z0,tool0\WObj:=Tableros;
    MoveL Target_2310,v100,z0,tool0\WObj:=Tableros;
  ENDPROC
  PROC Path_2A()
    MoveJ Target_2320,v200,z10,tool0\WObj:=Tableros;
    MoveL Target_2330,v100,z0,tool0\WObj:=Tableros;
    MoveL Target_2340,v100,z0,tool0\WObj:=Tableros;
    MoveL Target_2350,v100,z0,tool0\WObj:=Tableros;
    MoveL Target_2360,v100,z0,tool0\WObj:=Tableros;
    MoveL Target_2370,v100,z0,tool0\WObj:=Tableros;
    MoveL Target_2380,v100,z0,tool0\WObj:=Tableros;
    MoveL Target_2390,v100,z0,tool0\WObj:=Tableros;
    MoveL Target_2400,v100,z0,tool0\WObj:=Tableros;
    MoveL Target_2410,v100,z0,tool0\WObj:=Tableros;
    MoveL Target_2420,v100,z0,tool0\WObj:=Tableros;
    MoveL Target_2430,v100,z0,tool0\WObj:=Tableros;
    MoveL Target_2440,v100,z0,tool0\WObj:=Tableros;
    MoveL Target_2450,v100,z0,tool0\WObj:=Tableros;
    MoveL Target_2460,v100,z0,tool0\WObj:=Tableros;
    MoveL Target_2470,v100,z0,tool0\WObj:=Tableros;
  ENDPROC
  PROC Path_2T()
    MoveJ Target_2480,v200,z10,tool0\WObj:=Tableros;
    MoveL Target_2490,v100,z0,tool0\WObj:=Tableros;
    MoveL Target_2500,v100,z0,tool0\WObj:=Tableros;
    MoveL Target_2510,v100,z0,tool0\WObj:=Tableros;
    MoveL Target_2520,v100,z0,tool0\WObj:=Tableros;
    MoveL Target_2530,v100,z0,tool0\WObj:=Tableros;
    MoveL Target_2540,v100,z0,tool0\WObj:=Tableros;
    MoveL Target_2550,v100,z0,tool0\WObj:=Tableros;
    MoveL Target_2560,v100,z0,tool0\WObj:=Tableros;
    MoveL Target_2570,v100,z0,tool0\WObj:=Tableros;
    MoveL Target_2580,v100,z0,tool0\WObj:=Tableros;
  ENDPROC
  PROC Path_31()
    MoveJ Target_2590,v200,z10,tool0\WObj:=Tableros;
    MoveL Target_2600,v100,z0,tool0\WObj:=Tableros;
    MoveL Target_2610,v100,z0,tool0\WObj:=Tableros;
    MoveL Target_2620,v100,z0,tool0\WObj:=Tableros;
    MoveL Target_2630,v100,z0,tool0\WObj:=Tableros;
    MoveC Target_2640,Target_2650,v100,z0,tool0\WObj:=Tableros;
    MoveC Target_2660,Target_2670,v100,z0,tool0\WObj:=Tableros;
    MoveC Target_2680,Target_2690,v100,z0,tool0\WObj:=Tableros;
    MoveC Target_2700,Target_2710,v100,z0,tool0\WObj:=Tableros;
    MoveL Target_2720,v100,z0,tool0\WObj:=Tableros;
    MoveL Target_2730,v100,z0,tool0\WObj:=Tableros;
    MoveL Target_2740,v100,z0,tool0\WObj:=Tableros;
    MoveC Target_2750,Target_2760,v100,z0,tool0\WObj:=Tableros;
    MoveC Target_2770,Target_2780,v100,z0,tool0\WObj:=Tableros;
    MoveC Target_2790,Target_2800,v100,z0,tool0\WObj:=Tableros;
    MoveC Target_2810,Target_2820,v100,z0,tool0\WObj:=Tableros;
    MoveL Target_2830,v100,z0,tool0\WObj:=Tableros;
  ENDPROC
  PROC Path_32()
    MoveJ Target_2890,v200,z10,tool0\WObj:=Tableros;
    MoveL Target_2900,v100,z0,tool0\WObj:=Tableros;
    MoveC Target_2910,Target_2920,v100,z0,tool0\WObj:=Tableros;
    MoveC Target_2930,Target_2940,v100,z0,tool0\WObj:=Tableros;
    MoveL Target_2950,v100,z0,tool0\WObj:=Tableros;
  ENDPROC
ENDMODULE


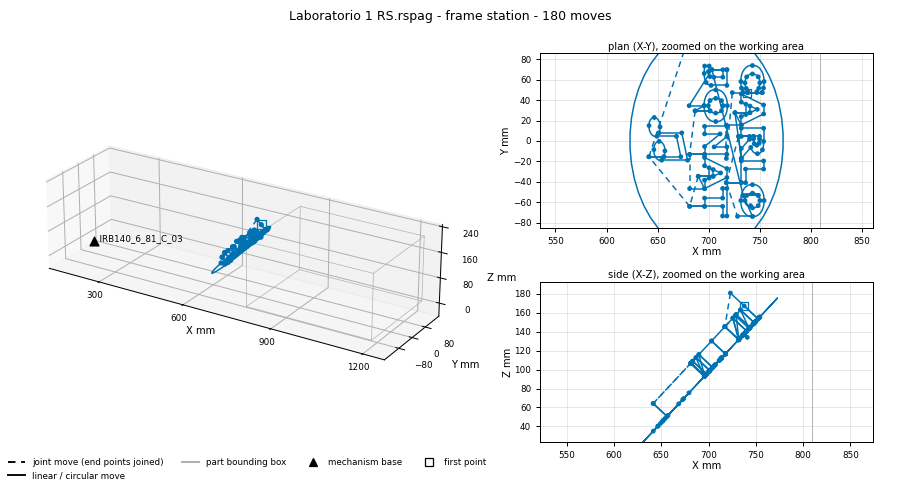
[picture p0: tool path of Laboratorio 1 RS.rspag in frame station, 180 of 180 moves have a stored position in this frame; points joined in program order, loops and branches not executed]
--- Controller Data/IRB140_6_81/RAPID/TASK1/PROGMOD/ModuleDecoCJ.mod ---
MODULE ModuleDecoCJ
    TASK PERS tooldata MarcadorTCP:=[TRUE,[[65.542,0,135.848],[0.974839064,0,0.222909847,0]],[1,[0,0,1],[1,0,0,0],0,0,0]];
    TASK PERS wobjdata Tableros:=[FALSE,TRUE,"",[[-164.785633838,0,0],[1,0,0,0]],[[800,-150,204.695],[0.398545746,0,0.917148455,0]]];
    CONST robtarget Target_350_2:=[[69.849,197.313,-20],[1,0,0,0],[0,0,0,0],[9E+09,9E+09,9E+09,9E+09,9E+09,9E+09]];
    CONST robtarget Target_360_2:=[[69.849,197.313,0],[1,0,0,0],[0,0,0,0],[9E+09,9E+09,9E+09,9E+09,9E+09,9E+09]];
    CONST robtarget Target_370_2:=[[68.877,199.4,0],[1,0,0,0],[0,0,0,0],[9E+09,9E+09,9E+09,9E+09,9E+09,9E+09]];
    CONST robtarget Target_380_2:=[[67.982,201.773,0],[1,0,0,0],[0,0,0,0],[9E+09,9E+09,9E+09,9E+09,9E+09,9E+09]];
    CONST robtarget Target_390_2:=[[67.399,204.703,0],[1,0,0,0],[0,0,0,0],[9E+09,9E+09,9E+09,9E+09,9E+09,9E+09]];
    CONST robtarget Target_400_2:=[[67.178,208.126,0],[1,0,0,0],[0,0,0,0],[9E+09,9E+09,9E+09,9E+09,9E+09,9E+09]];
    CONST robtarget Target_410_2:=[[71.703,219.575,0],[1,0,0,0],[0,0,0,0],[9E+09,9E+09,9E+09,9E+09,9E+09,9E+09]];
    CONST robtarget Target_420_2:=[[83.827,223.815,0],[1,0,0,0],[0,0,0,0],[9E+09,9E+09,9E+09,9E+09,9E+09,9E+09]];
    CONST robtarget Target_430_2:=[[96.066,219.588,0],[1,0,0,0],[0,0,0,0],[9E+09,9E+09,9E+09,9E+09,9E+09,9E+09]];
    CONST robtarget Target_440_2:=[[100.423,208.152,0],[1,0,0,0],[0,0,0,0],[9E+09,9E+09,9E+09,9E+09,9E+09,9E+09]];
    CONST robtarget Target_450_2:=[[100.19,204.561,0],[1,0,0,0],[0,0,0,0],[9E+09,9E+09,9E+09,9E+09,9E+09,9E+09]];
    CONST robtarget Target_460_2:=[[99.489,201.747,0],[1,0,0,0],[0,0,0,0],[9E+09,9E+09,9E+09,9E+09,9E+09,9E+09]];
    CONST robtarget Target_470_2:=[[98.608,199.348,0],[1,0,0,0],[0,0,0,0],[9E+09,9E+09,9E+09,9E+09,9E+09,9E+09]];
    CONST robtarget Target_480_2:=[[97.674,197.313,0],[1,0,0,0],[0,0,0,0],[9E+09,9E+09,9E+09,9E+09,9E+09,9E+09]];
    CONST robtarget Target_490_2:=[[90.154,197.313,0],[1,0,0,0],[0,0,0,0],[9E+09,9E+09,9E+09,9E+09,9E+09,9E+09]];
    CONST robtarget Target_500_2:=[[90.154,198.039,0],[1,0,0,0],[0,0,0,0],[9E+09,9E+09,9E+09,9E+09,9E+09,9E+09]];
    CONST robtarget Target_510_2:=[[91.386,199.452,0],[1,0,0,0],[0,0,0,0],[9E+09,9E+09,9E+09,9E+09,9E+09,9E+09]];
    CONST robtarget Target_520_2:=[[92.721,201.358,0],[1,0,0,0],[0,0,0,0],[9E+09,9E+09,9E+09,9E+09,9E+09,9E+09]];
    CONST robtarget Target_530_2:=[[93.901,203.783,0],[1,0,0,0],[0,0,0,0],[9E+09,9E+09,9E+09,9E+09,9E+09,9E+09]];
    CONST robtarget Target_540_2:=[[94.433,206.804,0],[1,0,0,0],[0,0,0,0],[9E+09,9E+09,9E+09,9E+09,9E+09,9E+09]];
    CONST robtarget Target_550_2:=[[93.901,209.864,0],[1,0,0,0],[0,0,0,0],[9E+09,9E+09,9E+09,9E+09,9E+09,9E+09]];
    CONST robtarget Target_560_2:=[[92.151,212.639,0],[1,0,0,0],[0,0,0,0],[9E+09,9E+09,9E+09,9E+09,9E+09,9E+09]];
    CONST robtarget Target_570_2:=[[88.87,214.726,0],[1,0,0,0],[0,0,0,0],[9E+09,9E+09,9E+09,9E+09,9E+09,9E+09]];
    CONST robtarget Target_580_2:=[[83.852,215.517,0],[1,0,0,0],[0,0,0,0],[9E+09,9E+09,9E+09,9E+09,9E+09,9E+09]];
    CONST robtarget Target_590_2:=[[78.938,214.752,0],[1,0,0,0],[0,0,0,0],[9E+09,9E+09,9E+09,9E+09,9E+09,9E+09]];
    CONST robtarget Target_600_2:=[[75.632,212.794,0],[1,0,0,0],[0,0,0,0],[9E+09,9E+09,9E+09,9E+09,9E+09,9E+09]];
    CONST robtarget Target_610_2:=[[73.713,210.032,0],[1,0,0,0],[0,0,0,0],[9E+09,9E+09,9E+09,9E+09,9E+09,9E+09]];
    CONST robtarget Target_620_2:=[[73.169,206.856,0],[1,0,0,0],[0,0,0,0],[9E+09,9E+09,9E+09,9E+09,9E+09,9E+09]];
    CONST robtarget Target_630_2:=[[73.648,204.042,0],[1,0,0,0],[0,0,0,0],[9E+09,9E+09,9E+09,9E+09,9E+09,9E+09]];
    CONST robtarget Target_640_2:=[[74.828,201.592,0],[1,0,0,0],[0,0,0,0],[9E+09,9E+09,9E+09,9E+09,9E+09,9E+09]];
    CONST robtarget Target_650_2:=[[76.228,199.595,0],[1,0,0,0],[0,0,0,0],[9E+09,9E+09,9E+09,9E+09,9E+09,9E+09]];
    CONST robtarget Target_660_2:=[[77.473,198.117,0],[1,0,0,0],[0,0,0,0],[9E+09,9E+09,9E+09,9E+09,9E+09,9E+09]];
    CONST robtarget Target_670_2:=[[77.473,197.313,0],[1,0,0,0],[0,0,0,0],[9E+09,9E+09,9E+09,9E+09,9E+09,9E+09]];
    CONST robtarget Target_680_2:=[[69.849,197.313,0],[1,0,0,0],[0,0,0,0],[9E+09,9E+09,9E+09,9E+09,9E+09,9E+09]];
    CONST robtarget Target_690_2:=[[69.849,197.313,-40],[1,0,0,0],[0,0,0,0],[9E+09,9E+09,9E+09,9E+09,9E+09,9E+09]];
    CONST robtarget Target_1010_2:=[[99.801,132.872,-20],[1,0,0,0],[0,0,0,0],[9E+09,9E+09,9E+09,9E+09,9E+09,9E+09]];
    CONST robtarget Target_850_2:=[[99.801,165.624,-20],[1,0,0,0],[0,0,0,0],[9E+09,9E+09,9E+09,9E+09,9E+09,9E+09]];
    CONST robtarget Target_860_2:=[[99.801,165.624,0],[1,0,0,0],[0,0,0,0],[9E+09,9E+09,9E+09,9E+09,9E+09,9E+09]];
    CONST robtarget Target_870_2:=[[67.801,176.438,0],[1,0,0,0],[0,0,0,0],[9E+09,9E+09,9E+09,9E+09,9E+09,9E+09]];
    CONST robtarget Target_880_2:=[[67.801,185.203,0],[1,0,0,0],[0,0,0,0],[9E+09,9E+09,9E+09,9E+09,9E+09,9E+09]];
    CONST robtarget Target_890_2:=[[99.801,196.016,0],[1,0,0,0],[0,0,0,0],[9E+09,9E+09,9E+09,9E+09,9E+09,9E+09]];
    CONST robtarget Target_900_2:=[[99.801,187.977,0],[1,0,0,0],[0,0,0,0],[9E+09,9E+09,9E+09,9E+09,9E+09,9E+09]];
    CONST robtarget Target_910_2:=[[93.266,185.955,0],[1,0,0,0],[0,0,0,0],[9E+09,9E+09,9E+09,9E+09,9E+09,9E+09]];
    CONST robtarget Target_920_2:=[[93.266,175.893,0],[1,0,0,0],[0,0,0,0],[9E+09,9E+09,9E+09,9E+09,9E+09,9E+09]];
    CONST robtarget Target_930_2:=[[99.801,173.896,0],[1,0,0,0],[0,0,0,0],[9E+09,9E+09,9E+09,9E+09,9E+09,9E+09]];
    CONST robtarget Target_940_2:=[[99.801,165.624,0],[1,0,0,0],[0,0,0,0],[9E+09,9E+09,9E+09,9E+09,9E+09,9E+09]];
    CONST robtarget Target_950_2:=[[87.457,177.656,-20],[1,0,0,0],[0,0,0,0],[9E+09,9E+09,9E+09,9E+09,9E+09,9E+09]];
    CONST robtarget Target_960_2:=[[87.457,177.656,0],[1,0,0,0],[0,0,0,0],[9E+09,9E+09,9E+09,9E+09,9E+09,9E+09]];
    CONST robtarget Target_970_2:=[[76.877,180.924,0],[1,0,0,0],[0,0,0,0],[9E+09,9E+09,9E+09,9E+09,9E+09,9E+09]];
    CONST robtarget Target_980_2:=[[87.457,184.217,0],[1,0,0,0],[0,0,0,0],[9E+09,9E+09,9E+09,9E+09,9E+09,9E+09]];
    CONST robtarget Target_990_2:=[[87.457,177.656,0],[1,0,0,0],[0,0,0,0],[9E+09,9E+09,9E+09,9E+09,9E+09,9E+09]];
    CONST robtarget Target_1000_2:=[[87.457,177.656,-20],[1,0,0,0],[0,0,0,0],[9E+09,9E+09,9E+09,9E+09,9E+09,9E+09]];
    CONST robtarget Target_1020_2:=[[99.801,132.872,0],[1,0,0,0],[0,0,0,0],[9E+09,9E+09,9E+09,9E+09,9E+09,9E+09]];
    CONST robtarget Target_1030_2:=[[86.186,143.634,0],[1,0,0,0],[0,0,0,0],[9E+09,9E+09,9E+09,9E+09,9E+09,9E+09]];
    CONST robtarget Target_1040_2:=[[82.543,139.199,0],[1,0,0,0],[0,0,0,0],[9E+09,9E+09,9E+09,9E+09,9E+09,9E+09]];
    CONST robtarget Target_1050_2:=[[76.592,137.54,0],[1,0,0,0],[0,0,0,0],[9E+09,9E+09,9E+09,9E+09,9E+09,9E+09]];
    CONST robtarget Target_1060_2:=[[72.3,138.551,0],[1,0,0,0],[0,0,0,0],[9E+09,9E+09,9E+09,9E+09,9E+09,9E+09]];
    CONST robtarget Target_1070_2:=[[69.512,141.274,0],[1,0,0,0],[0,0,0,0],[9E+09,9E+09,9E+09,9E+09,9E+09,9E+09]];
    CONST robtarget Target_1080_2:=[[68.138,144.93,0],[1,0,0,0],[0,0,0,0],[9E+09,9E+09,9E+09,9E+09,9E+09,9E+09]];
    CONST robtarget Target_1090_2:=[[67.801,149.572,0],[1,0,0,0],[0,0,0,0],[9E+09,9E+09,9E+09,9E+09,9E+09,9E+09]];
    CONST robtarget Target_1100_2:=[[67.801,162.434,0],[1,0,0,0],[0,0,0,0],[9E+09,9E+09,9E+09,9E+09,9E+09,9E+09]];
    CONST robtarget Target_1110_2:=[[99.801,162.434,0],[1,0,0,0],[0,0,0,0],[9E+09,9E+09,9E+09,9E+09,9E+09,9E+09]];
    CONST robtarget Target_1120_2:=[[99.801,154.447,0],[1,0,0,0],[0,0,0,0],[9E+09,9E+09,9E+09,9E+09,9E+09,9E+09]];
    CONST robtarget Target_1130_2:=[[88.053,154.447,0],[1,0,0,0],[0,0,0,0],[9E+09,9E+09,9E+09,9E+09,9E+09,9E+09]];
    CONST robtarget Target_1140_2:=[[88.053,151.543,0],[1,0,0,0],[0,0,0,0],[9E+09,9E+09,9E+09,9E+09,9E+09,9E+09]];
    CONST robtarget Target_1150_2:=[[99.801,142.648,0],[1,0,0,0],[0,0,0,0],[9E+09,9E+09,9E+09,9E+09,9E+09,9E+09]];
    CONST robtarget Target_1160_2:=[[99.801,132.872,0],[1,0,0,0],[0,0,0,0],[9E+09,9E+09,9E+09,9E+09,9E+09,9E+09]];
    CONST robtarget Target_1170_2:=[[82.297,154.447,-20],[1,0,0,0],[0,0,0,0],[9E+09,9E+09,9E+09,9E+09,9E+09,9E+09]];
    CONST robtarget Target_1180_2:=[[82.297,154.447,0],[1,0,0,0],[0,0,0,0],[9E+09,9E+09,9E+09,9E+09,9E+09,9E+09]];
    CONST robtarget Target_1190_2:=[[82.297,152.139,0],[1,0,0,0],[0,0,0,0],[9E+09,9E+09,9E+09,9E+09,9E+09,9E+09]];
    CONST robtarget Target_1200_2:=[[82.089,149.3,0],[1,0,0,0],[0,0,0,0],[9E+09,9E+09,9E+09,9E+09,9E+09,9E+09]];
    CONST robtarget Target_1210_2:=[[81.233,147.316,0],[1,0,0,0],[0,0,0,0],[9E+09,9E+09,9E+09,9E+09,9E+09,9E+09]];
    CONST robtarget Target_1220_2:=[[79.781,146.162,0],[1,0,0,0],[0,0,0,0],[9E+09,9E+09,9E+09,9E+09,9E+09,9E+09]];
    CONST robtarget Target_1230_2:=[[77.603,145.786,0],[1,0,0,0],[0,0,0,0],[9E+09,9E+09,9E+09,9E+09,9E+09,9E+09]];
    CONST robtarget Target_1240_2:=[[75.515,146.253,0],[1,0,0,0],[0,0,0,0],[9E+09,9E+09,9E+09,9E+09,9E+09,9E+09]];
    CONST robtarget Target_1250_2:=[[74.18,147.783,0],[1,0,0,0],[0,0,0,0],[9E+09,9E+09,9E+09,9E+09,9E+09,9E+09]];
    CONST robtarget Target_1260_2:=[[73.778,149.455,0],[1,0,0,0],[0,0,0,0],[9E+09,9E+09,9E+09,9E+09,9E+09,9E+09]];
    CONST robtarget Target_1270_2:=[[73.687,151.75,0],[1,0,0,0],[0,0,0,0],[9E+09,9E+09,9E+09,9E+09,9E+09,9E+09]];
    CONST robtarget Target_1280_2:=[[73.687,154.447,0],[1,0,0,0],[0,0,0,0],[9E+09,9E+09,9E+09,9E+09,9E+09,9E+09]];
    CONST robtarget Target_1290_2:=[[82.297,154.447,0],[1,0,0,0],[0,0,0,0],[9E+09,9E+09,9E+09,9E+09,9E+09,9E+09]];
    CONST robtarget Target_1300_2:=[[82.297,154.447,-20],[1,0,0,0],[0,0,0,0],[9E+09,9E+09,9E+09,9E+09,9E+09,9E+09]];
    CONST robtarget Target_1310_2:=[[99.801,109.144,-20],[1,0,0,0],[0,0,0,0],[9E+09,9E+09,9E+09,9E+09,9E+09,9E+09]];
    CONST robtarget Target_1320_2:=[[99.801,109.144,0],[1,0,0,0],[0,0,0,0],[9E+09,9E+09,9E+09,9E+09,9E+09,9E+09]];
    CONST robtarget Target_1330_2:=[[93.707,109.144,0],[1,0,0,0],[0,0,0,0],[9E+09,9E+09,9E+09,9E+09,9E+09,9E+09]];
    CONST robtarget Target_1340_2:=[[93.707,122.447,0],[1,0,0,0],[0,0,0,0],[9E+09,9E+09,9E+09,9E+09,9E+09,9E+09]];
    CONST robtarget Target_1350_2:=[[67.801,122.447,0],[1,0,0,0],[0,0,0,0],[9E+09,9E+09,9E+09,9E+09,9E+09,9E+09]];
    CONST robtarget Target_1360_2:=[[67.801,130.486,0],[1,0,0,0],[0,0,0,0],[9E+09,9E+09,9E+09,9E+09,9E+09,9E+09]];
    CONST robtarget Target_1370_2:=[[99.801,130.486,0],[1,0,0,0],[0,0,0,0],[9E+09,9E+09,9E+09,9E+09,9E+09,9E+09]];
    CONST robtarget Target_1380_2:=[[99.801,109.144,0],[1,0,0,0],[0,0,0,0],[9E+09,9E+09,9E+09,9E+09,9E+09,9E+09]];
    CONST robtarget Target_1390_2:=[[99.801,109.144,-20],[1,0,0,0],[0,0,0,0],[9E+09,9E+09,9E+09,9E+09,9E+09,9E+09]];
    CONST robtarget Target_1400_2:=[[83.801,76.185,-20],[1,0,0,0],[0,0,0,0],[9E+09,9E+09,9E+09,9E+09,9E+09,9E+09]];
    CONST robtarget Target_1410_2:=[[83.801,76.185,0],[1,0,0,0],[0,0,0,0],[9E+09,9E+09,9E+09,9E+09,9E+09,9E+09]];
    CONST robtarget Target_1420_2:=[[96.028,80.334,0],[1,0,0,0],[0,0,0,0],[9E+09,9E+09,9E+09,9E+09,9E+09,9E+09]];
    CONST robtarget Target_1430_2:=[[100.475,91.692,0],[1,0,0,0],[0,0,0,0],[9E+09,9E+09,9E+09,9E+09,9E+09,9E+09]];
    CONST robtarget Target_1440_2:=[[95.976,103.05,0],[1,0,0,0],[0,0,0,0],[9E+09,9E+09,9E+09,9E+09,9E+09,9E+09]];
    CONST robtarget Target_1450_2:=[[83.801,107.173,0],[1,0,0,0],[0,0,0,0],[9E+09,9E+09,9E+09,9E+09,9E+09,9E+09]];
    CONST robtarget Target_1460_2:=[[71.613,103.05,0],[1,0,0,0],[0,0,0,0],[9E+09,9E+09,9E+09,9E+09,9E+09,9E+09]];
    CONST robtarget Target_1470_2:=[[67.126,91.692,0],[1,0,0,0],[0,0,0,0],[9E+09,9E+09,9E+09,9E+09,9E+09,9E+09]];
    CONST robtarget Target_1480_2:=[[71.587,80.334,0],[1,0,0,0],[0,0,0,0],[9E+09,9E+09,9E+09,9E+09,9E+09,9E+09]];
    CONST robtarget Target_1490_2:=[[83.801,76.185,0],[1,0,0,0],[0,0,0,0],[9E+09,9E+09,9E+09,9E+09,9E+09,9E+09]];
    CONST robtarget Target_1500_2:=[[75.58,96.671,-20],[1,0,0,0],[0,0,0,0],[9E+09,9E+09,9E+09,9E+09,9E+09,9E+09]];
    CONST robtarget Target_1510_2:=[[75.58,96.671,0],[1,0,0,0],[0,0,0,0],[9E+09,9E+09,9E+09,9E+09,9E+09,9E+09]];
    CONST robtarget Target_1520_2:=[[78.887,98.266,0],[1,0,0,0],[0,0,0,0],[9E+09,9E+09,9E+09,9E+09,9E+09,9E+09]];
    CONST robtarget Target_1530_2:=[[83.801,98.875,0],[1,0,0,0],[0,0,0,0],[9E+09,9E+09,9E+09,9E+09,9E+09,9E+09]];
    CONST robtarget Target_1540_2:=[[88.702,98.292,0],[1,0,0,0],[0,0,0,0],[9E+09,9E+09,9E+09,9E+09,9E+09,9E+09]];
    CONST robtarget Target_1550_2:=[[91.969,96.697,0],[1,0,0,0],[0,0,0,0],[9E+09,9E+09,9E+09,9E+09,9E+09,9E+09]];
    CONST robtarget Target_1560_2:=[[93.862,94.376,0],[1,0,0,0],[0,0,0,0],[9E+09,9E+09,9E+09,9E+09,9E+09,9E+09]];
    CONST robtarget Target_1570_2:=[[94.433,91.666,0],[1,0,0,0],[0,0,0,0],[9E+09,9E+09,9E+09,9E+09,9E+09,9E+09]];
    CONST robtarget Target_1580_2:=[[93.823,88.917,0],[1,0,0,0],[0,0,0,0],[9E+09,9E+09,9E+09,9E+09,9E+09,9E+09]];
    CONST robtarget Target_1590_2:=[[91.917,86.635,5],[1,0,0,0],[0,0,0,0],[9E+09,9E+09,9E+09,9E+09,9E+09,9E+09]];
    CONST robtarget Target_1600_2:=[[88.663,85.041,0],[1,0,0,0],[0,0,0,0],[9E+09,9E+09,9E+09,9E+09,9E+09,9E+09]];
    CONST robtarget Target_1610_2:=[[83.801,84.483,0],[1,0,0,0],[0,0,0,0],[9E+09,9E+09,9E+09,9E+09,9E+09,9E+09]];
    CONST robtarget Target_1620_2:=[[78.912,85.066,0],[1,0,0,0],[0,0,0,0],[9E+09,9E+09,9E+09,9E+09,9E+09,9E+09]];
    CONST robtarget Target_1630_2:=[[75.632,86.661,0],[1,0,0,0],[0,0,0,0],[9E+09,9E+09,9E+09,9E+09,9E+09,9E+09]];
    CONST robtarget Target_1640_2:=[[73.739,88.969,0],[1,0,0,0],[0,0,0,0],[9E+09,9E+09,9E+09,9E+09,9E+09,9E+09]];
    CONST robtarget Target_1650_2:=[[73.169,91.666,0],[1,0,0,0],[0,0,0,0],[9E+09,9E+09,9E+09,9E+09,9E+09,9E+09]];
    CONST robtarget Target_1660_2:=[[73.7,94.35,0],[1,0,0,0],[0,0,0,0],[9E+09,9E+09,9E+09,9E+09,9E+09,9E+09]];
    CONST robtarget Target_1670_2:=[[75.58,96.671,0],[1,0,0,0],[0,0,0,0],[9E+09,9E+09,9E+09,9E+09,9E+09,9E+09]];
    CONST robtarget Target_1680_2:=[[75.58,96.671,-20],[1,0,0,0],[0,0,0,0],[9E+09,9E+09,9E+09,9E+09,9E+09,9E+09]];
    CONST robtarget Target_1690_2:=[[120.488,219.705,-20],[1,0,0,0],[0,0,0,0],[9E+09,9E+09,9E+09,9E+09,9E+09,9E+09]];
    CONST robtarget Target_1700_2:=[[120.488,219.705,0],[1,0,0,0],[0,0,0,0],[9E+09,9E+09,9E+09,9E+09,9E+09,9E+09]];
    CONST robtarget Target_1710_2:=[[120.488,204.353,0],[1,0,0,0],[0,0,0,0],[9E+09,9E+09,9E+09,9E+09,9E+09,9E+09]];
    CONST robtarget Target_1720_2:=[[143.1,204.353,0.001],[1,0,0,0],[0,0,0,0],[9E+09,9E+09,9E+09,9E+09,9E+09,9E+09]];
    CONST robtarget Target_1730_2:=[[147.016,205.066,0.001],[1,0,0,0],[0,0,0,0],[9E+09,9E+09,9E+09,9E+09,9E+09,9E+09]];
    CONST robtarget Target_1740_2:=[[150.154,207.206,0.001],[1,0,0,0],[0,0,0,0],[9E+09,9E+09,9E+09,9E+09,9E+09,9E+09]];
    CONST robtarget Target_1750_2:=[[152.293,211.005,0.001],[1,0,0,0],[0,0,0,0],[9E+09,9E+09,9E+09,9E+09,9E+09,9E+09]];
    CONST robtarget Target_1760_2:=[[152.98,216.049,0.001],[1,0,0,0],[0,0,0,0],[9E+09,9E+09,9E+09,9E+09,9E+09,9E+09]];
    CONST robtarget Target_1770_2:=[[152.825,220.042,0.001],[1,0,0,0],[0,0,0,0],[9E+09,9E+09,9E+09,9E+09,9E+09,9E+09]];
    CONST robtarget Target_1780_2:=[[152.358,223.335,0.001],[1,0,0,0],[0,0,0,0],[9E+09,9E+09,9E+09,9E+09,9E+09,9E+09]];
    CONST robtarget Target_1790_2:=[[145.875,223.335,0.001],[1,0,0,0],[0,0,0,0],[9E+09,9E+09,9E+09,9E+09,9E+09,9E+09]];
    CONST robtarget Target_1800_2:=[[146.601,220.6,0.001],[1,0,0,0],[0,0,0,0],[9E+09,9E+09,9E+09,9E+09,9E+09,9E+09]];
    CONST robtarget Target_1810_2:=[[146.938,217.89,0.001],[1,0,0,0],[0,0,0,0],[9E+09,9E+09,9E+09,9E+09,9E+09,9E+09]];
    CONST robtarget Target_1820_2:=[[146.342,214.609,0.001],[1,0,0,0],[0,0,0,0],[9E+09,9E+09,9E+09,9E+09,9E+09,9E+09]];
    CONST robtarget Target_1830_2:=[[144.656,212.989,0.001],[1,0,0,0],[0,0,0,0],[9E+09,9E+09,9E+09,9E+09,9E+09,9E+09]];
    CONST robtarget Target_1840_2:=[[142.219,212.444,0.001],[1,0,0,0],[0,0,0,0],[9E+09,9E+09,9E+09,9E+09,9E+09,9E+09]];
    CONST robtarget Target_1850_2:=[[139.133,212.392,0],[1,0,0,0],[0,0,0,0],[9E+09,9E+09,9E+09,9E+09,9E+09,9E+09]];
    CONST robtarget Target_1860_2:=[[126.297,212.392,0],[1,0,0,0],[0,0,0,0],[9E+09,9E+09,9E+09,9E+09,9E+09,9E+09]];
    CONST robtarget Target_1870_2:=[[126.297,219.705,0],[1,0,0,0],[0,0,0,0],[9E+09,9E+09,9E+09,9E+09,9E+09,9E+09]];
    CONST robtarget Target_1880_2:=[[120.488,219.705,0],[1,0,0,0],[0,0,0,0],[9E+09,9E+09,9E+09,9E+09,9E+09,9E+09]];
    CONST robtarget Target_1890_2:=[[120.488,219.705,-20],[1,0,0,0],[0,0,0,0],[9E+09,9E+09,9E+09,9E+09,9E+09,9E+09]];
    CONST robtarget Target_1900_2:=[[153.162,184.515,-20],[1,0,0,0],[0,0,0,0],[9E+09,9E+09,9E+09,9E+09,9E+09,9E+09]];
    CONST robtarget Target_1910_2:=[[153.162,184.515,0],[1,0,0,0],[0,0,0,0],[9E+09,9E+09,9E+09,9E+09,9E+09,9E+09]];
    CONST robtarget Target_1920_2:=[[148.715,173.157,0.001],[1,0,0,0],[0,0,0,0],[9E+09,9E+09,9E+09,9E+09,9E+09,9E+09]];
    CONST robtarget Target_1930_2:=[[136.488,169.008,0],[1,0,0,0],[0,0,0,0],[9E+09,9E+09,9E+09,9E+09,9E+09,9E+09]];
    CONST robtarget Target_1940_2:=[[124.274,173.157,0],[1,0,0,0],[0,0,0,0],[9E+09,9E+09,9E+09,9E+09,9E+09,9E+09]];
    CONST robtarget Target_1950_2:=[[119.814,184.515,0],[1,0,0,0],[0,0,0,0],[9E+09,9E+09,9E+09,9E+09,9E+09,9E+09]];
    CONST robtarget Target_1960_2:=[[124.3,195.874,0],[1,0,0,0],[0,0,0,0],[9E+09,9E+09,9E+09,9E+09,9E+09,9E+09]];
    CONST robtarget Target_1970_2:=[[136.488,199.997,0],[1,0,0,0],[0,0,0,0],[9E+09,9E+09,9E+09,9E+09,9E+09,9E+09]];
    CONST robtarget Target_1980_2:=[[148.663,195.874,0.001],[1,0,0,0],[0,0,0,0],[9E+09,9E+09,9E+09,9E+09,9E+09,9E+09]];
    CONST robtarget Target_1990_2:=[[153.162,184.515,0.001],[1,0,0,0],[0,0,0,0],[9E+09,9E+09,9E+09,9E+09,9E+09,9E+09]];
    CONST robtarget Target_2000_2:=[[144.604,179.459,-20],[1,0,0,0],[0,0,0,0],[9E+09,9E+09,9E+09,9E+09,9E+09,9E+09]];
    CONST robtarget Target_2010_2:=[[144.604,179.459,0.001],[1,0,0,0],[0,0,0,0],[9E+09,9E+09,9E+09,9E+09,9E+09,9E+09]];
    CONST robtarget Target_2020_2:=[[141.35,177.864,0.001],[1,0,0,0],[0,0,0,0],[9E+09,9E+09,9E+09,9E+09,9E+09,9E+09]];
    CONST robtarget Target_2030_2:=[[136.488,177.306,0],[1,0,0,0],[0,0,0,0],[9E+09,9E+09,9E+09,9E+09,9E+09,9E+09]];
    CONST robtarget Target_2040_2:=[[131.6,177.89,0],[1,0,0,0],[0,0,0,0],[9E+09,9E+09,9E+09,9E+09,9E+09,9E+09]];
    CONST robtarget Target_2050_2:=[[128.319,179.485,0],[1,0,0,0],[0,0,0,0],[9E+09,9E+09,9E+09,9E+09,9E+09,9E+09]];
    CONST robtarget Target_2060_2:=[[126.426,181.793,0],[1,0,0,0],[0,0,0,0],[9E+09,9E+09,9E+09,9E+09,9E+09,9E+09]];
    CONST robtarget Target_2070_2:=[[125.856,184.489,0],[1,0,0,0],[0,0,0,0],[9E+09,9E+09,9E+09,9E+09,9E+09,9E+09]];
    CONST robtarget Target_2080_2:=[[126.387,187.173,0],[1,0,0,0],[0,0,0,0],[9E+09,9E+09,9E+09,9E+09,9E+09,9E+09]];
    CONST robtarget Target_2090_2:=[[128.267,189.494,0],[1,0,0,0],[0,0,0,0],[9E+09,9E+09,9E+09,9E+09,9E+09,9E+09]];
    CONST robtarget Target_2100_2:=[[131.574,191.089,0],[1,0,0,0],[0,0,0,0],[9E+09,9E+09,9E+09,9E+09,9E+09,9E+09]];
    CONST robtarget Target_2110_2:=[[136.488,191.699,0],[1,0,0,0],[0,0,0,0],[9E+09,9E+09,9E+09,9E+09,9E+09,9E+09]];
    CONST robtarget Target_2120_2:=[[141.389,191.115,0.001],[1,0,0,0],[0,0,0,0],[9E+09,9E+09,9E+09,9E+09,9E+09,9E+09]];
    CONST robtarget Target_2130_2:=[[144.656,189.52,0.001],[1,0,0,0],[0,0,0,0],[9E+09,9E+09,9E+09,9E+09,9E+09,9E+09]];
    CONST robtarget Target_2140_2:=[[146.549,187.199,0.001],[1,0,0,0],[0,0,0,0],[9E+09,9E+09,9E+09,9E+09,9E+09,9E+09]];
    CONST robtarget Target_2150_2:=[[147.12,184.489,0.001],[1,0,0,0],[0,0,0,0],[9E+09,9E+09,9E+09,9E+09,9E+09,9E+09]];
    CONST robtarget Target_2160_2:=[[146.51,181.741,0.001],[1,0,0,0],[0,0,0,0],[9E+09,9E+09,9E+09,9E+09,9E+09,9E+09]];
    CONST robtarget Target_2170_2:=[[144.604,179.459,0.001],[1,0,0,0],[0,0,0,0],[9E+09,9E+09,9E+09,9E+09,9E+09,9E+09]];
    CONST robtarget Target_2180_2:=[[144.604,179.459,-20],[1,0,0,0],[0,0,0,0],[9E+09,9E+09,9E+09,9E+09,9E+09,9E+09]];
    CONST robtarget Target_2190_2:=[[152.488,136.827,-20],[1,0,0,0],[0,0,0,0],[9E+09,9E+09,9E+09,9E+09,9E+09,9E+09]];
    CONST robtarget Target_2200_2:=[[152.488,136.827,0.001],[1,0,0,0],[0,0,0,0],[9E+09,9E+09,9E+09,9E+09,9E+09,9E+09]];
    CONST robtarget Target_2210_2:=[[120.488,136.827,0],[1,0,0,0],[0,0,0,0],[9E+09,9E+09,9E+09,9E+09,9E+09,9E+09]];
    CONST robtarget Target_2220_2:=[[120.488,144.165,0],[1,0,0,0],[0,0,0,0],[9E+09,9E+09,9E+09,9E+09,9E+09,9E+09]];
    CONST robtarget Target_2230_2:=[[138.822,144.165,0],[1,0,0,0],[0,0,0,0],[9E+09,9E+09,9E+09,9E+09,9E+09,9E+09]];
    CONST robtarget Target_2240_2:=[[120.488,154.382,0],[1,0,0,0],[0,0,0,0],[9E+09,9E+09,9E+09,9E+09,9E+09,9E+09]];
    CONST robtarget Target_2250_2:=[[120.488,164.237,0],[1,0,0,0],[0,0,0,0],[9E+09,9E+09,9E+09,9E+09,9E+09,9E+09]];
    CONST robtarget Target_2260_2:=[[152.488,164.237,0.001],[1,0,0,0],[0,0,0,0],[9E+09,9E+09,9E+09,9E+09,9E+09,9E+09]];
    CONST robtarget Target_2270_2:=[[152.488,156.898,0.001],[1,0,0,0],[0,0,0,0],[9E+09,9E+09,9E+09,9E+09,9E+09,9E+09]];
    CONST robtarget Target_2280_2:=[[130.186,156.898,0],[1,0,0,0],[0,0,0,0],[9E+09,9E+09,9E+09,9E+09,9E+09,9E+09]];
    CONST robtarget Target_2290_2:=[[152.488,144.554,0.001],[1,0,0,0],[0,0,0,0],[9E+09,9E+09,9E+09,9E+09,9E+09,9E+09]];
    CONST robtarget Target_2300_2:=[[152.488,136.827,0.001],[1,0,0,0],[0,0,0,0],[9E+09,9E+09,9E+09,9E+09,9E+09,9E+09]];
    CONST robtarget Target_2310_2:=[[152.488,136.827,-20],[1,0,0,0],[0,0,0,0],[9E+09,9E+09,9E+09,9E+09,9E+09,9E+09]];
    CONST robtarget Target_2320_2:=[[152.488,103.374,-20],[1,0,0,0],[0,0,0,0],[9E+09,9E+09,9E+09,9E+09,9E+09,9E+09]];
    CONST robtarget Target_2330_2:=[[152.488,103.374,0.001],[1,0,0,0],[0,0,0,0],[9E+09,9E+09,9E+09,9E+09,9E+09,9E+09]];
    CONST robtarget Target_2340_2:=[[120.488,114.188,0],[1,0,0,0],[0,0,0,0],[9E+09,9E+09,9E+09,9E+09,9E+09,9E+09]];
    CONST robtarget Target_2350_2:=[[120.488,122.953,0],[1,0,0,0],[0,0,0,0],[9E+09,9E+09,9E+09,9E+09,9E+09,9E+09]];
    CONST robtarget Target_2360_2:=[[152.488,133.767,0.001],[1,0,0,0],[0,0,0,0],[9E+09,9E+09,9E+09,9E+09,9E+09,9E+09]];
    CONST robtarget Target_2370_2:=[[152.488,125.728,0.001],[1,0,0,0],[0,0,0,0],[9E+09,9E+09,9E+09,9E+09,9E+09,9E+09]];
    CONST robtarget Target_2380_2:=[[145.953,123.705,0.001],[1,0,0,0],[0,0,0,0],[9E+09,9E+09,9E+09,9E+09,9E+09,9E+09]];
    CONST robtarget Target_2390_2:=[[145.953,113.643,0.001],[1,0,0,0],[0,0,0,0],[9E+09,9E+09,9E+09,9E+09,9E+09,9E+09]];
    CONST robtarget Target_2400_2:=[[152.488,111.647,0.001],[1,0,0,0],[0,0,0,0],[9E+09,9E+09,9E+09,9E+09,9E+09,9E+09]];
    CONST robtarget Target_2410_2:=[[152.488,103.374,0.001],[1,0,0,0],[0,0,0,0],[9E+09,9E+09,9E+09,9E+09,9E+09,9E+09]];
    CONST robtarget Target_2420_2:=[[140.144,115.407,-20],[1,0,0,0],[0,0,0,0],[9E+09,9E+09,9E+09,9E+09,9E+09,9E+09]];
    CONST robtarget Target_2430_2:=[[140.144,115.407,0.001],[1,0,0,0],[0,0,0,0],[9E+09,9E+09,9E+09,9E+09,9E+09,9E+09]];
    CONST robtarget Target_2440_2:=[[129.564,118.674,0],[1,0,0,0],[0,0,0,0],[9E+09,9E+09,9E+09,9E+09,9E+09,9E+09]];
    CONST robtarget Target_2450_2:=[[140.144,121.968,0.001],[1,0,0,0],[0,0,0,0],[9E+09,9E+09,9E+09,9E+09,9E+09,9E+09]];
    CONST robtarget Target_2460_2:=[[140.144,115.407,0.001],[1,0,0,0],[0,0,0,0],[9E+09,9E+09,9E+09,9E+09,9E+09,9E+09]];
    CONST robtarget Target_2470_2:=[[140.144,115.407,-20],[1,0,0,0],[0,0,0,0],[9E+09,9E+09,9E+09,9E+09,9E+09,9E+09]];
    CONST robtarget Target_2480_2:=[[152.488,86,-20],[1,0,0,0],[0,0,0,0],[9E+09,9E+09,9E+09,9E+09,9E+09,9E+09]];
    CONST robtarget Target_2490_2:=[[152.488,86,0.001],[1,0,0,0],[0,0,0,0],[9E+09,9E+09,9E+09,9E+09,9E+09,9E+09]];
    CONST robtarget Target_2500_2:=[[126.582,86,0],[1,0,0,0],[0,0,0,0],[9E+09,9E+09,9E+09,9E+09,9E+09,9E+09]];
    CONST robtarget Target_2510_2:=[[126.582,76.535,0],[1,0,0,0],[0,0,0,0],[9E+09,9E+09,9E+09,9E+09,9E+09,9E+09]];
    CONST robtarget Target_2520_2:=[[120.488,76.535,0],[1,0,0,0],[0,0,0,0],[9E+09,9E+09,9E+09,9E+09,9E+09,9E+09]];
    CONST robtarget Target_2530_2:=[[120.488,103.504,0],[1,0,0,0],[0,0,0,0],[9E+09,9E+09,9E+09,9E+09,9E+09,9E+09]];
    CONST robtarget Target_2540_2:=[[126.582,103.504,0],[1,0,0,0],[0,0,0,0],[9E+09,9E+09,9E+09,9E+09,9E+09,9E+09]];
    CONST robtarget Target_2550_2:=[[126.582,94.039,0],[1,0,0,0],[0,0,0,0],[9E+09,9E+09,9E+09,9E+09,9E+09,9E+09]];
    CONST robtarget Target_2560_2:=[[152.488,94.039,0.001],[1,0,0,0],[0,0,0,0],[9E+09,9E+09,9E+09,9E+09,9E+09,9E+09]];
    CONST robtarget Target_2570_2:=[[152.488,86,0.001],[1,0,0,0],[0,0,0,0],[9E+09,9E+09,9E+09,9E+09,9E+09,9E+09]];
    CONST robtarget Target_2580_2:=[[152.488,86,-20],[1,0,0,0],[0,0,0,0],[9E+09,9E+09,9E+09,9E+09,9E+09,9E+09]];
    CONST robtarget Target_2590_2:=[[210.888,134.542,-20],[1,0,0,0],[0,0,0,0],[9E+09,9E+09,9E+09,9E+09,9E+09,9E+09]];
    CONST robtarget Target_2600_2:=[[210.888,134.542,0.001],[1,0,0,0],[0,0,0,0],[9E+09,9E+09,9E+09,9E+09,9E+09,9E+09]];
    CONST robtarget Target_2610_2:=[[186.577,134.542,0.001],[1,0,0,0],[0,0,0,0],[9E+09,9E+09,9E+09,9E+09,9E+09,9E+09]];
    CONST robtarget Target_2620_2:=[[192.776,154.518,0.001],[1,0,0,0],[0,0,0,0],[9E+09,9E+09,9E+09,9E+09,9E+09,9E+09]];
    CONST robtarget Target_2630_2:=[[220.856,154.518,0.001],[1,0,0,0],[0,0,0,0],[9E+09,9E+09,9E+09,9E+09,9E+09,9E+09]];
    CONST robtarget Target_2640_2:=[[229.253,157.086,0.001],[1,0,0,0],[0,0,0,0],[9E+09,9E+09,9E+09,9E+09,9E+09,9E+09]];
    CONST robtarget Target_2650_2:=[[232.16,165.012,0.001],[1,0,0,0],[0,0,0,0],[9E+09,9E+09,9E+09,9E+09,9E+09,9E+09]];
    CONST robtarget Target_2660_2:=[[230.094,170.806,0.001],[1,0,0,0],[0,0,0,0],[9E+09,9E+09,9E+09,9E+09,9E+09,9E+09]];
    CONST robtarget Target_2670_2:=[[224.705,172.954,0.001],[1,0,0,0],[0,0,0,0],[9E+09,9E+09,9E+09,9E+09,9E+09,9E+09]];
    CONST robtarget Target_2680_2:=[[218.789,170.401,0.001],[1,0,0,0],[0,0,0,0],[9E+09,9E+09,9E+09,9E+09,9E+09,9E+09]];
    CONST robtarget Target_2690_2:=[[216.399,163.716,0.001],[1,0,0,0],[0,0,0,0],[9E+09,9E+09,9E+09,9E+09,9E+09,9E+09]];
    CONST robtarget Target_2700_2:=[[216.784,160.94,0.001],[1,0,0,0],[0,0,0,0],[9E+09,9E+09,9E+09,9E+09,9E+09,9E+09]];
    CONST robtarget Target_2710_2:=[[217.938,157.881,0.001],[1,0,0,0],[0,0,0,0],[9E+09,9E+09,9E+09,9E+09,9E+09,9E+09]];
    CONST robtarget Target_2720_2:=[[185.159,157.881,0.001],[1,0,0,0],[0,0,0,0],[9E+09,9E+09,9E+09,9E+09,9E+09,9E+09]];
    CONST robtarget Target_2730_2:=[[176.852,131.139,0.001],[1,0,0,0],[0,0,0,0],[9E+09,9E+09,9E+09,9E+09,9E+09,9E+09]];
    CONST robtarget Target_2740_2:=[[214.048,131.139,0.001],[1,0,0,0],[0,0,0,0],[9E+09,9E+09,9E+09,9E+09,9E+09,9E+09]];
    CONST robtarget Target_2750_2:=[[222.254,133.615,0.001],[1,0,0,0],[0,0,0,0],[9E+09,9E+09,9E+09,9E+09,9E+09,9E+09]];
    CONST robtarget Target_2760_2:=[[225.191,141.511,0.001],[1,0,0,0],[0,0,0,0],[9E+09,9E+09,9E+09,9E+09,9E+09,9E+09]];
    CONST robtarget Target_2770_2:=[[223.084,147.346,0.001],[1,0,0,0],[0,0,0,0],[9E+09,9E+09,9E+09,9E+09,9E+09,9E+09]];
    CONST robtarget Target_2780_2:=[[217.655,149.534,0.001],[1,0,0,0],[0,0,0,0],[9E+09,9E+09,9E+09,9E+09,9E+09,9E+09]];
    CONST robtarget Target_2790_2:=[[211.86,146.941,0.001],[1,0,0,0],[0,0,0,0],[9E+09,9E+09,9E+09,9E+09,9E+09,9E+09]];
    CONST robtarget Target_2800_2:=[[209.429,140.255,0.001],[1,0,0,0],[0,0,0,0],[9E+09,9E+09,9E+09,9E+09,9E+09,9E+09]];
    CONST robtarget Target_2810_2:=[[209.672,137.905,0.001],[1,0,0,0],[0,0,0,0],[9E+09,9E+09,9E+09,9E+09,9E+09,9E+09]];
    CONST robtarget Target_2820_2:=[[210.888,134.542,0.001],[1,0,0,0],[0,0,0,0],[9E+09,9E+09,9E+09,9E+09,9E+09,9E+09]];
    CONST robtarget Target_2830_2:=[[210.888,134.542,-20],[1,0,0,0],[0,0,0,0],[9E+09,9E+09,9E+09,9E+09,9E+09,9E+09]];
    CONST robtarget Target_2890_2:=[[149.643,260,-20],[1,0,0,0],[0,0,0,0],[9E+09,9E+09,9E+09,9E+09,9E+09,9E+09]];
    CONST robtarget Target_2900_2:=[[149.643,260,0.001],[1,0,0,0],[0,0,0,0],[9E+09,9E+09,9E+09,9E+09,9E+09,9E+09]];
    CONST robtarget Target_2910_2:=[[43.169,122.373,0],[1,0,0,0],[0,0,0,0],[9E+09,9E+09,9E+09,9E+09,9E+09,9E+09]];
    CONST robtarget Target_2920_2:=[[149.643,40,0.001],[1,0,0,0],[0,0,0,0],[9E+09,9E+09,9E+09,9E+09,9E+09,9E+09]];
    CONST robtarget Target_2930_2:=[[258.691,135.554,0.001],[1,0,0,0],[0,0,0,0],[9E+09,9E+09,9E+09,9E+09,9E+09,9E+09]];
    CONST robtarget Target_2940_2:=[[149.643,260,0.001],[1,0,0,0],[0,0,0,0],[9E+09,9E+09,9E+09,9E+09,9E+09,9E+09]];
    CONST robtarget Target_2950_2:=[[149.643,260,-20],[1,0,0,0],[0,0,0,0],[9E+09,9E+09,9E+09,9E+09,9E+09,9E+09]];
    LOCAL PROC Path_DecoComp()
        MoveJ Target_350_2,v200,z10,MarcadorTCP\WObj:=Tableros;
        MoveL Target_360_2,v100,z0,MarcadorTCP\WObj:=Tableros;
        MoveC Target_370_2,Target_380_2,v100,z0,MarcadorTCP\WObj:=Tableros;
        MoveC Target_390_2,Target_400_2,v100,z0,MarcadorTCP\WObj:=Tableros;
        MoveC Target_410_2,Target_420_2,v100,z0,MarcadorTCP\WObj:=Tableros;
        MoveC Target_430_2,Target_440_2,v100,z0,MarcadorTCP\WObj:=Tableros;
        MoveC Target_450_2,Target_460_2,v100,z0,MarcadorTCP\WObj:=Tableros;
        MoveC Target_470_2,Target_480_2,v100,z0,MarcadorTCP\WObj:=Tableros;
        MoveL Target_490_2,v100,z0,MarcadorTCP\WObj:=Tableros;
        MoveL Target_500_2,v100,z0,MarcadorTCP\WObj:=Tableros;
        MoveC Target_510_2,Target_520_2,v100,z0,MarcadorTCP\WObj:=Tableros;
        MoveC Target_530_2,Target_540_2,v100,z0,MarcadorTCP\WObj:=Tableros;
        MoveC Target_550_2,Target_560_2,v100,z0,MarcadorTCP\WObj:=Tableros;
        MoveC Target_570_2,Target_580_2,v100,z0,MarcadorTCP\WObj:=Tableros;
        MoveC Target_590_2,Target_600_2,v100,z0,MarcadorTCP\WObj:=Tableros;
        MoveC Target_610_2,Target_620_2,v100,z0,MarcadorTCP\WObj:=Tableros;
        MoveC Target_630_2,Target_640_2,v100,z0,MarcadorTCP\WObj:=Tableros;
        MoveC Target_650_2,Target_660_2,v100,z0,MarcadorTCP\WObj:=Tableros;
        MoveL Target_670_2,v100,z0,MarcadorTCP\WObj:=Tableros;
        MoveL Target_680_2,v100,z0,MarcadorTCP\WObj:=Tableros;
        MoveL Target_690_2,v100,z0,MarcadorTCP\WObj:=Tableros;
        MoveJ Target_1010_2,v200,z10,MarcadorTCP\WObj:=Tableros;
        MoveJ Target_850_2,v100,z10,MarcadorTCP\WObj:=Tableros;
        MoveL Target_860_2,v100,z0,MarcadorTCP\WObj:=Tableros;
        MoveL Target_870_2,v100,z0,MarcadorTCP\WObj:=Tableros;
        MoveL Target_880_2,v100,z0,MarcadorTCP\WObj:=Tableros;
        MoveL Target_890_2,v100,z0,MarcadorTCP\WObj:=Tableros;
        MoveL Target_900_2,v100,z0,MarcadorTCP\WObj:=Tableros;
        MoveL Target_910_2,v100,z0,MarcadorTCP\WObj:=Tableros;
        MoveL Target_920_2,v100,z0,MarcadorTCP\WObj:=Tableros;
        MoveL Target_930_2,v100,z0,MarcadorTCP\WObj:=Tableros;
        MoveL Target_940_2,v100,z0,MarcadorTCP\WObj:=Tableros;
        MoveL Target_950_2,v100,z0,MarcadorTCP\WObj:=Tableros;
        MoveL Target_960_2,v100,z0,MarcadorTCP\WObj:=Tableros;
        MoveL Target_970_2,v100,z0,MarcadorTCP\WObj:=Tableros;
        MoveL Target_980_2,v100,z0,MarcadorTCP\WObj:=Tableros;
        MoveL Target_990_2,v100,z0,MarcadorTCP\WObj:=Tableros;
        MoveL Target_1000_2,v100,z0,MarcadorTCP\WObj:=Tableros;
        MoveL Target_1020_2,v100,z0,MarcadorTCP\WObj:=Tableros;
        MoveL Target_1030_2,v100,z0,MarcadorTCP\WObj:=Tableros;
        MoveC Target_1040_2,Target_1050_2,v100,z0,MarcadorTCP\WObj:=Tableros;
        MoveC Target_1060_2,Target_1070_2,v100,z0,MarcadorTCP\WObj:=Tableros;
        MoveC Target_1080_2,Target_1090_2,v100,z0,MarcadorTCP\WObj:=Tableros;
        MoveL Target_1100_2,v100,z0,MarcadorTCP\WObj:=Tableros;
        MoveL Target_1110_2,v100,z0,MarcadorTCP\WObj:=Tableros;
        MoveL Target_1120_2,v100,z0,MarcadorTCP\WObj:=Tableros;
        MoveL Target_1130_2,v100,z0,MarcadorTCP\WObj:=Tableros;
        MoveL Target_1140_2,v100,z0,MarcadorTCP\WObj:=Tableros;
        MoveL Target_1150_2,v100,z0,MarcadorTCP\WObj:=Tableros;
        MoveL Target_1160_2,v100,z0,MarcadorTCP\WObj:=Tableros;
        MoveL Target_1170_2,v100,z0,MarcadorTCP\WObj:=Tableros;
        MoveL Target_1180_2,v100,z0,MarcadorTCP\WObj:=Tableros;
        MoveL Target_1190_2,v100,z0,MarcadorTCP\WObj:=Tableros;
        MoveC Target_1200_2,Target_1210_2,v100,z0,MarcadorTCP\WObj:=Tableros;
        MoveC Target_1220_2,Target_1230_2,v100,z0,MarcadorTCP\WObj:=Tableros;
        MoveC Target_1240_2,Target_1250_2,v100,z0,MarcadorTCP\WObj:=Tableros;
        MoveC Target_1260_2,Target_1270_2,v100,z0,MarcadorTCP\WObj:=Tableros;
        MoveL Target_1280_2,v100,z0,MarcadorTCP\WObj:=Tableros;
        MoveL Target_1290_2,v100,z0,MarcadorTCP\WObj:=Tableros;
        MoveL Target_1300_2,v100,z0,MarcadorTCP\WObj:=Tableros;
        MoveJ Target_1310_2,v200,z10,MarcadorTCP\WObj:=Tableros;
        MoveL Target_1320_2,v100,z0,MarcadorTCP\WObj:=Tableros;
        MoveL Target_1330_2,v100,z0,MarcadorTCP\WObj:=Tableros;
        MoveL Target_1340_2,v100,z0,MarcadorTCP\WObj:=Tableros;
        MoveL Target_1350_2,v100,z0,MarcadorTCP\WObj:=Tableros;
        MoveL Target_1360_2,v100,z0,MarcadorTCP\WObj:=Tableros;
        MoveL Target_1370_2,v100,z0,MarcadorTCP\WObj:=Tableros;
        MoveL Target_1380_2,v100,z0,MarcadorTCP\WObj:=Tableros;
        MoveL Target_1390_2,v100,z0,MarcadorTCP\WObj:=Tableros;
        MoveJ Target_1400_2,v200,z10,MarcadorTCP\WObj:=Tableros;
        MoveL Target_1410_2,v100,z0,MarcadorTCP\WObj:=Tableros;
        MoveC Target_1420_2,Target_1430_2,v100,z0,MarcadorTCP\WObj:=Tableros;
        MoveC Target_1440_2,Target_1450_2,v100,z0,MarcadorTCP\WObj:=Tableros;
        MoveC Target_1460_2,Target_1470_2,v100,z0,MarcadorTCP\WObj:=Tableros;
        MoveC Target_1480_2,Target_1490_2,v100,z0,MarcadorTCP\WObj:=Tableros;
        MoveL Target_1500_2,v100,z0,MarcadorTCP\WObj:=Tableros;
        MoveL Target_1510_2,v100,z0,MarcadorTCP\WObj:=Tableros;
        MoveC Target_1520_2,Target_1530_2,v100,z0,MarcadorTCP\WObj:=Tableros;
        MoveC Target_1540_2,Target_1550_2,v100,z0,MarcadorTCP\WObj:=Tableros;
        MoveC Target_1560_2,Target_1570_2,v100,z0,MarcadorTCP\WObj:=Tableros;
        MoveC Target_1580_2,Target_1590_2,v100,z0,MarcadorTCP\WObj:=Tableros;
        MoveC Target_1600_2,Target_1610_2,v100,z0,MarcadorTCP\WObj:=Tableros;
        MoveC Target_1620_2,Target_1630_2,v100,z0,MarcadorTCP\WObj:=Tableros;
        MoveC Target_1640_2,Target_1650_2,v100,z0,MarcadorTCP\WObj:=Tableros;
        MoveC Target_1660_2,Target_1670_2,v100,z0,MarcadorTCP\WObj:=Tableros;
        MoveL Target_1680_2,v100,z0,MarcadorTCP\WObj:=Tableros;
        MoveL Target_1690_2,v100,z0,MarcadorTCP\WObj:=Tableros;
        MoveL Target_1700_2,v100,z0,MarcadorTCP\WObj:=Tableros;
        MoveL Target_1710_2,v100,z0,MarcadorTCP\WObj:=Tableros;
        MoveL Target_1720_2,v100,z0,MarcadorTCP\WObj:=Tableros;
        MoveC Target_1730_2,Target_1740_2,v100,z0,MarcadorTCP\WObj:=Tableros;
        MoveC Target_1750_2,Target_1760_2,v100,z0,MarcadorTCP\WObj:=Tableros;
        MoveC Target_1770_2,Target_1780_2,v100,z0,MarcadorTCP\WObj:=Tableros;
        MoveL Target_1790_2,v100,z0,MarcadorTCP\WObj:=Tableros;
        MoveC Target_1800_2,Target_1810_2,v100,z0,MarcadorTCP\WObj:=Tableros;
        MoveC Target_1820_2,Target_1830_2,v100,z0,MarcadorTCP\WObj:=Tableros;
        MoveC Target_1840_2,Target_1850_2,v100,z0,MarcadorTCP\WObj:=Tableros;
        MoveL Target_1860_2,v100,z0,MarcadorTCP\WObj:=Tableros;
        MoveL Target_1870_2,v100,z0,MarcadorTCP\WObj:=Tableros;
        MoveL Target_1880_2,v100,z0,MarcadorTCP\WObj:=Tableros;
        MoveL Target_1890_2,v100,z0,MarcadorTCP\WObj:=Tableros;
        MoveL Target_1900_2,v100,z0,MarcadorTCP\WObj:=Tableros;
        MoveL Target_1910_2,v100,z0,MarcadorTCP\WObj:=Tableros;
        MoveC Target_1920_2,Target_1930_2,v100,z0,MarcadorTCP\WObj:=Tableros;
        MoveC Target_1940_2,Target_1950_2,v100,z0,MarcadorTCP\WObj:=Tableros;
        MoveC Target_1960_2,Target_1970_2,v100,z0,MarcadorTCP\WObj:=Tableros;
        MoveC Target_1980_2,Target_1990_2,v100,z0,MarcadorTCP\WObj:=Tableros;
        MoveL Target_2000_2,v100,z0,MarcadorTCP\WObj:=Tableros;
        MoveL Target_2010_2,v100,z0,MarcadorTCP\WObj:=Tableros;
        MoveC Target_2020_2,Target_2030_2,v100,z0,MarcadorTCP\WObj:=Tableros;
        MoveC Target_2040_2,Target_2050_2,v100,z0,MarcadorTCP\WObj:=Tableros;
        MoveC Target_2060_2,Target_2070_2,v100,z0,MarcadorTCP\WObj:=Tableros;
        MoveC Target_2080_2,Target_2090_2,v100,z0,MarcadorTCP\WObj:=Tableros;
        MoveC Target_2100_2,Target_2110_2,v100,z0,MarcadorTCP\WObj:=Tableros;
        MoveC Target_2120_2,Target_2130_2,v100,z0,MarcadorTCP\WObj:=Tableros;
        MoveC Target_2140_2,Target_2150_2,v100,z0,MarcadorTCP\WObj:=Tableros;
        MoveC Target_2160_2,Target_2170_2,v100,z0,MarcadorTCP\WObj:=Tableros;
        MoveL Target_2180_2,v100,z0,MarcadorTCP\WObj:=Tableros;
        MoveJ Target_2190_2,v200,z10,MarcadorTCP\WObj:=Tableros;
        MoveL Target_2200_2,v100,z0,MarcadorTCP\WObj:=Tableros;
        MoveL Target_2210_2,v100,z0,MarcadorTCP\WObj:=Tableros;
        MoveL Target_2220_2,v100,z0,MarcadorTCP\WObj:=Tableros;
        MoveL Target_2230_2,v100,z0,MarcadorTCP\WObj:=Tableros;
        MoveL Target_2240_2,v100,z0,MarcadorTCP\WObj:=Tableros;
        MoveL Target_2250_2,v100,z0,MarcadorTCP\WObj:=Tableros;
        MoveL Target_2260_2,v100,z0,MarcadorTCP\WObj:=Tableros;
        MoveL Target_2270_2,v100,z0,MarcadorTCP\WObj:=Tableros;
        MoveL Target_2280_2,v100,z0,MarcadorTCP\WObj:=Tableros;
        MoveL Target_2290_2,v100,z0,MarcadorTCP\WObj:=Tableros;
        MoveL Target_2300_2,v100,z0,MarcadorTCP\WObj:=Tableros;
        MoveL Target_2310_2,v100,z0,MarcadorTCP\WObj:=Tableros;
        MoveJ Target_2320_2,v200,z10,MarcadorTCP\WObj:=Tableros;
        MoveL Target_2330_2,v100,z0,MarcadorTCP\WObj:=Tableros;
        MoveL Target_2340_2,v100,z0,MarcadorTCP\WObj:=Tableros;
        MoveL Target_2350_2,v100,z0,MarcadorTCP\WObj:=Tableros;
        MoveL Target_2360_2,v100,z0,MarcadorTCP\WObj:=Tableros;
        MoveL Target_2370_2,v100,z0,MarcadorTCP\WObj:=Tableros;
        MoveL Target_2380_2,v100,z0,MarcadorTCP\WObj:=Tableros;
        MoveL Target_2390_2,v100,z0,MarcadorTCP\WObj:=Tableros;
        MoveL Target_2400_2,v100,z0,MarcadorTCP\WObj:=Tableros;
        MoveL Target_2410_2,v100,z0,MarcadorTCP\WObj:=Tableros;
        MoveL Target_2420_2,v100,z0,MarcadorTCP\WObj:=Tableros;
        MoveL Target_2430_2,v100,z0,MarcadorTCP\WObj:=Tableros;
        MoveL Target_2440_2,v100,z0,MarcadorTCP\WObj:=Tableros;
        MoveL Target_2450_2,v100,z0,MarcadorTCP\WObj:=Tableros;
        MoveL Target_2460_2,v100,z0,MarcadorTCP\WObj:=Tableros;
        MoveL Target_2470_2,v100,z0,MarcadorTCP\WObj:=Tableros;
        MoveJ Target_2480_2,v200,z10,MarcadorTCP\WObj:=Tableros;
        MoveL Target_2490_2,v100,z0,MarcadorTCP\WObj:=Tableros;
        MoveL Target_2500_2,v100,z0,MarcadorTCP\WObj:=Tableros;
        MoveL Target_2510_2,v100,z0,MarcadorTCP\WObj:=Tableros;
        MoveL Target_2520_2,v100,z0,MarcadorTCP\WObj:=Tableros;
        MoveL Target_2530_2,v100,z0,MarcadorTCP\WObj:=Tableros;
        MoveL Target_2540_2,v100,z0,MarcadorTCP\WObj:=Tableros;
        MoveL Target_2550_2,v100,z0,MarcadorTCP\WObj:=Tableros;
        MoveL Target_2560_2,v100,z0,MarcadorTCP\WObj:=Tableros;
        MoveL Target_2570_2,v100,z0,MarcadorTCP\WObj:=Tableros;
        MoveL Target_2580_2,v100,z0,MarcadorTCP\WObj:=Tableros;
        MoveJ Target_2590_2,v200,z10,MarcadorTCP\WObj:=Tableros;
        MoveL Target_2600_2,v100,z0,MarcadorTCP\WObj:=Tableros;
        MoveL Target_2610_2,v100,z0,MarcadorTCP\WObj:=Tableros;
        MoveL Target_2620_2,v100,z0,MarcadorTCP\WObj:=Tableros;
        MoveL Target_2630_2,v100,z0,MarcadorTCP\WObj:=Tableros;
        MoveC Target_2640_2,Target_2650_2,v100,z0,MarcadorTCP\WObj:=Tableros;
        MoveC Target_2660_2,Target_2670_2,v100,z0,MarcadorTCP\WObj:=Tableros;
        MoveC Target_2680_2,Target_2690_2,v100,z0,MarcadorTCP\WObj:=Tableros;
        MoveC Target_2700_2,Target_2710_2,v100,z0,MarcadorTCP\WObj:=Tableros;
        MoveL Target_2720_2,v100,z0,MarcadorTCP\WObj:=Tableros;
        MoveL Target_2730_2,v100,z0,MarcadorTCP\WObj:=Tableros;
        MoveL Target_2740_2,v100,z0,MarcadorTCP\WObj:=Tableros;
        MoveC Target_2750_2,Target_2760_2,v100,z0,MarcadorTCP\WObj:=Tableros;
        MoveC Target_2770_2,Target_2780_2,v100,z0,MarcadorTCP\WObj:=Tableros;
        MoveC Target_2790_2,Target_2800_2,v100,z0,MarcadorTCP\WObj:=Tableros;
        MoveC Target_2810_2,Target_2820_2,v100,z0,MarcadorTCP\WObj:=Tableros;
        MoveL Target_2830_2,v100,z0,MarcadorTCP\WObj:=Tableros;
        MoveJ Target_2890_2,v200,z10,MarcadorTCP\WObj:=Tableros;
        MoveL Target_2900_2,v100,z0,MarcadorTCP\WObj:=Tableros;
        MoveC Target_2910_2,Target_2920_2,v100,z0,MarcadorTCP\WObj:=Tableros;
        MoveC Target_2930_2,Target_2940_2,v100,z0,MarcadorTCP\WObj:=Tableros;
        MoveL Target_2950_2,v100,z0,MarcadorTCP\WObj:=Tableros;
    ENDPROC
ENDMODULE
